LIN {X 0,Y 474.686,Z 210.351,A -85,B 0,C 180,E1 -7391.963,E2 -7391.963} C_VEL
LIN {X 0,Y 474.649,Z 210.356,A -85,B 0,C 180,E1 -7395.778,E2 -7395.778} C_VEL
LIN {X 0,Y 474.614,Z 210.365,A -85,B 0,C 180,E1 -7399.012,E2 -7399.012} C_VEL
LIN {X 0,Y 474.547,Z 210.369,A -85,B 0,C 180,E1 -7401.731,E2 -7401.731} C_VEL
LIN {X 0,Y 474.613,Z 210.367,A -85,B 0,C 180,E1 -7404.495,E2 -7404.495} C_VEL
LIN {X 0,Y 474.635,Z 210.358,A -85,B 0,C 180,E1 -7407.337,E2 -7407.337} C_VEL
LIN {X 0,Y 474.56,Z 210.372,A -85,B 0,C 180,E1 -7410.813,E2 -7410.813} C_VEL
LIN {X 0,Y 474.597,Z 210.364,A -85,B 0,C 180,E1 -7413.987,E2 -7413.987} C_VEL
LIN {X 0,Y 474.534,Z 210.373,A -85,B 0,C 180,E1 -7416.903,E2 -7416.903} C_VEL
LIN {X 0,Y 474.58,Z 210.365,A -85,B 0,C 180,E1 -7419.649,E2 -7419.649} C_VEL
LIN {X 0,Y 474.589,Z 210.37,A -85,B 0,C 180,E1 -7422.24,E2 -7422.24} C_VEL
LIN {X 0,Y 474.584,Z 210.364,A -85,B 0,C 180,E1 -7425.301,E2 -7425.301} C_VEL
LIN {X 0,Y 474.591,Z 210.371,A -85,B 0,C 180,E1 -7428.218,E2 -7428.218} C_VEL
LIN {X 0,Y 474.617,Z 210.365,A -85,B 0,C 180,E1 -7430.458,E2 -7430.458} C_VEL
LIN {X 0,Y 474.568,Z 210.368,A -85,B 0,C 180,E1 -7433.68,E2 -7433.68} C_VEL
LIN {X 0,Y 474.621,Z 210.36,A -85,B 0,C 180,E1 -7436.783,E2 -7436.783} C_VEL
LIN {X 0,Y 474.586,Z 210.368,A -85,B 0,C 180,E1 -7439.773,E2 -7439.773} C_VEL
LIN {X 0,Y 474.681,Z 210.353,A -85,B 0,C 180,E1 -7442.683,E2 -7442.683} C_VEL
LIN {X 0,Y 474.627,Z 210.361,A -85,B 0,C 180,E1 -7445.509,E2 -7445.509} C_VEL
LIN {X 0,Y 474.659,Z 210.355,A -85,B 0,C 180,E1 -7449.188,E2 -7449.188} C_VEL
LIN {X 0,Y 474.634,Z 210.363,A -85,B 0,C 180,E1 -7451.707,E2 -7451.707} C_VEL
LIN {X 0,Y 473.967,Z 210.452,A -85,B 0,C 180,E1 -7452.416,E2 -7452.416} C_VEL
LIN {X 0,Y 471.117,Z 210.806,A -85,B 0,C 180,E1 -7453.568,E2 -7453.568} C_VEL
LIN {X 0,Y 468.706,Z 211.101,A -85,B 0,C 180,E1 -7454.496,E2 -7454.496} C_VEL
LIN {X 0,Y 467.669,Z 211.227,A -85,B 0,C 180,E1 -7455.213,E2 -7455.213} C_VEL
LIN {X 0,Y 467.583,Z 211.237,A -85,B 0,C 180,E1 -7455.456,E2 -7455.456} C_VEL
LIN {X 0,Y 467.645,Z 211.228,A -85,B 0,C 180,E1 -7458.736,E2 -7458.736} C_VEL
LIN {X 0,Y 467.666,Z 211.23,A -85,B 0,C 180,E1 -7461.359,E2 -7461.359} C_VEL
LIN {X 0,Y 467.718,Z 211.227,A -85,B 0,C 180,E1 -7463.964,E2 -7463.964} C_VEL
LIN {X 0,Y 467.696,Z 211.354,A -85,B 0,C 180,E1 -7465.099,E2 -7465.099} C_VEL
LIN {X 0,Y 468.519,Z 218.325,A -85,B 0,C 180,E1 -7466.562,E2 -7466.562} C_VEL
LIN {X 0,Y 468.443,Z 226.016,A -85,B 0,C 180,E1 -7468.121,E2 -7468.121} C_VEL
LIN {X 0,Y 471.287,Z 240.784,A -85,B 0,C 180,E1 -7468.453,E2 -7468.453} C_VEL
LIN {X 0,Y 470.521,Z 333.446,A -85,B 0,C 180,E1 -7469.895,E2 -7469.895} C_VEL
LIN {X 0,Y 470.229,Z 346.46,A -85,B 0,C 180,E1 -7470.269,E2 -7470.269} C_VEL
LIN {X 0,Y 469.945,Z 358.958,A -85,B 0,C 180,E1 -7470.805,E2 -7470.805} C_VEL
LIN {X 0,Y 469.51,Z 370.947,A -85,B 0,C 180,E1 -7471.502,E2 -7471.502} C_VEL
LIN {X 0,Y 468.954,Z 382.395,A -85,B 0,C 180,E1 -7472.363,E2 -7472.363} C_VEL
LIN {X 0,Y 468.529,Z 392.675,A -85,B 0,C 180,E1 -7473.333,E2 -7473.333} C_VEL
LIN {X 0,Y 468.097,Z 401.117,A -85,B 0,C 180,E1 -7474.306,E2 -7474.306} C_VEL
LIN {X 0,Y 467.694,Z 410.256,A -85,B 0,C 180,E1 -7475.606,E2 -7475.606} C_VEL
LIN {X 0,Y 467.398,Z 417.615,A -85,B 0,C 180,E1 -7476.91,E2 -7476.91} C_VEL
LIN {X 0,Y 467.126,Z 423.538,A -85,B 0,C 180,E1 -7478.218,E2 -7478.218} C_VEL
LIN {X 0,Y 466.911,Z 428.222,A -85,B 0,C 180,E1 -7479.531,E2 -7479.531} C_VEL
LIN {X 0,Y 466.795,Z 431.791,A -85,B 0,C 180,E1 -7480.848,E2 -7480.848} C_VEL
LIN {X 0,Y 466.701,Z 434.341,A -85,B 0,C 180,E1 -7482.171,E2 -7482.171} C_VEL
LIN {X 0,Y 466.604,Z 435.521,A -85,B 0,C 180,E1 -7483.058,E2 -7483.058} C_VEL
LIN {X 0,Y 466.58,Z 436.247,A -85,B 0,C 180,E1 -7483.946,E2 -7483.946} C_VEL
LIN {X 0,Y 466.616,Z 436.558,A -85,B 0,C 180,E1 -7485.433,E2 -7485.433} C_VEL
LIN {X 0,Y 466.566,Z 435.978,A -85,B 0,C 180,E1 -7486.631,E2 -7486.631} C_VEL
LIN {X 0,Y 466.628,Z 435.02,A -85,B 0,C 180,E1 -7487.531,E2 -7487.531} C_VEL
LIN {X 0,Y 466.737,Z 433.625,A -85,B 0,C 180,E1 -7488.444,E2 -7488.444} C_VEL
LIN {X 0,Y 466.862,Z 430.671,A -85,B 0,C 180,E1 -7489.798,E2 -7489.798} C_VEL
LIN {X 0,Y 467.026,Z 426.549,A -85,B 0,C 180,E1 -7491.171,E2 -7491.171} C_VEL
LIN {X 0,Y 467.303,Z 420.044,A -85,B 0,C 180,E1 -7492.784,E2 -7492.784} C_VEL
LIN {X 0,Y 467.679,Z 412.837,A -85,B 0,C 180,E1 -7494.172,E2 -7494.172} C_VEL
LIN {X 0,Y 468.058,Z 405.338,A -85,B 0,C 180,E1 -7495.336,E2 -7495.336} C_VEL
LIN {X 0,Y 468.534,Z 396.074,A -85,B 0,C 180,E1 -7496.502,E2 -7496.502} C_VEL
LIN {X 0,Y 469.022,Z 385.744,A -85,B 0,C 180,E1 -7497.557,E2 -7497.557} C_VEL
LIN {X 0,Y 469.553,Z 375.373,A -85,B 0,C 180,E1 -7498.407,E2 -7498.407} C_VEL
LIN {X 0,Y 470.036,Z 363.063,A -85,B 0,C 180,E1 -7499.196,E2 -7499.196} C_VEL
LIN {X 0,Y 470.43,Z 350.815,A -85,B 0,C 180,E1 -7499.784,E2 -7499.784} C_VEL
LIN {X 0,Y 470.664,Z 338.306,A -85,B 0,C 180,E1 -7500.211,E2 -7500.211} C_VEL
LIN {X 0,Y 470.823,Z 323.886,A -85,B 0,C 180,E1 -7500.497,E2 -7500.497} C_VEL
LIN {X 0,Y 471.613,Z 240.593,A -85,B 0,C 180,E1 -7501.782,E2 -7501.782} C_VEL
LIN {X 0,Y 468.664,Z 226.097,A -85,B 0,C 180,E1 -7502.147,E2 -7502.147} C_VEL
LIN {X 0,Y 468.703,Z 216.769,A -85,B 0,C 180,E1 -7504.025,E2 -7504.025} C_VEL
LIN {X 0,Y 467.613,Z 211.238,A -85,B 0,C 180,E1 -7505.221,E2 -7505.221} C_VEL
LIN {X 0,Y 467.564,Z 211.247,A -85,B 0,C 180,E1 -7508.592,E2 -7508.592} C_VEL
LIN {X 0,Y 467.577,Z 211.237,A -85,B 0,C 180,E1 -7511.4,E2 -7511.4} C_VEL
LIN {X 0,Y 467.561,Z 211.246,A -85,B 0,C 180,E1 -7513.822,E2 -7513.822} C_VEL
LIN {X 0,Y 467.595,Z 211.237,A -85,B 0,C 180,E1 -7517.441,E2 -7517.441} C_VEL
LIN {X 0,Y 467.581,Z 211.239,A -85,B 0,C 180,E1 -7520.856,E2 -7520.856} C_VEL
LIN {X 0,Y 467.543,Z 211.245,A -85,B 0,C 180,E1 -7524.259,E2 -7524.259} C_VEL
LIN {X 0,Y 467.561,Z 211.241,A -85,B 0,C 180,E1 -7527.32,E2 -7527.32} C_VEL
LIN {X 0,Y 467.553,Z 211.239,A -85,B 0,C 180,E1 -7530.665,E2 -7530.665} C_VEL
LIN {X 0,Y 467.592,Z 211.236,A -85,B 0,C 180,E1 -7533.198,E2 -7533.198} C_VEL
LIN {X 0,Y 467.573,Z 211.238,A -85,B 0,C 180,E1 -7536.466,E2 -7536.466} C_VEL
LIN {X 0,Y 467.598,Z 211.239,A -85,B 0,C 180,E1 -7539.776,E2 -7539.776} C_VEL
LIN {X 0,Y 467.584,Z 211.234,A -85,B 0,C 180,E1 -7542.506,E2 -7542.506} C_VEL
LIN {X 0,Y 467.579,Z 211.24,A -85,B 0,C 180,E1 -7545.196,E2 -7545.196} C_VEL
LIN {X 0,Y 467.626,Z 211.234,A -85,B 0,C 180,E1 -7547.854,E2 -7547.854} C_VEL
LIN {X 0,Y 467.653,Z 211.231,A -85,B 0,C 180,E1 -7551.357,E2 -7551.357} C_VEL
LIN {X 0,Y 467.725,Z 211.22,A -85,B 0,C 180,E1 -7553.963,E2 -7553.963} C_VEL
LIN {X 0,Y 467.827,Z 211.209,A -85,B 0,C 180,E1 -7557.417,E2 -7557.417} C_VEL
LIN {X 0,Y 467.846,Z 211.2,A -85,B 0,C 180,E1 -7560,E2 -7560} C_VEL
LIN {X 0,Y 467.826,Z 211.204,A -85,B 0,C 180,E1 -7562.583,E2 -7562.583} C_VEL
LIN {X 0,Y 467.697,Z 211.216,A -85,B 0,C 180,E1 -7566.038,E2 -7566.038} C_VEL
LIN {X 0,Y 467.64,Z 211.23,A -85,B 0,C 180,E1 -7568.644,E2 -7568.644} C_VEL
LIN {X 0,Y 467.654,Z 211.226,A -85,B 0,C 180,E1 -7572.146,E2 -7572.146} C_VEL
LIN {X 0,Y 467.62,Z 211.23,A -85,B 0,C 180,E1 -7575.885,E2 -7575.885} C_VEL
LIN {X 0,Y 467.594,Z 211.235,A -85,B 0,C 180,E1 -7579.309,E2 -7579.309} C_VEL
LIN {X 0,Y 467.504,Z 211.247,A -85,B 0,C 180,E1 -7582.076,E2 -7582.076} C_VEL
LIN {X 0,Y 467.542,Z 211.248,A -85,B 0,C 180,E1 -7584.891,E2 -7584.891} C_VEL
LIN {X 0,Y 467.557,Z 211.238,A -85,B 0,C 180,E1 -7587.773,E2 -7587.773} C_VEL
LIN {X 0,Y 467.529,Z 211.244,A -85,B 0,C 180,E1 -7591.043,E2 -7591.043} C_VEL
LIN {X 0,Y 467.557,Z 211.245,A -85,B 0,C 180,E1 -7594.242,E2 -7594.242} C_VEL
LIN {X 0,Y 467.523,Z 211.243,A -85,B 0,C 180,E1 -7597.187,E2 -7597.187} C_VEL
LIN {X 0,Y 467.554,Z 211.245,A -85,B 0,C 180,E1 -7600.267,E2 -7600.267} C_VEL
LIN {X 0,Y 467.547,Z 211.242,A -85,B 0,C 180,E1 -7602.565,E2 -7602.565} C_VEL
LIN {X 0,Y 467.553,Z 211.241,A -85,B 0,C 180,E1 -7605.054,E2 -7605.054} C_VEL
LIN {X 0,Y 467.557,Z 211.243,A -85,B 0,C 180,E1 -7608.598,E2 -7608.598} C_VEL
LIN {X 0,Y 467.556,Z 211.247,A -85,B 0,C 180,E1 -7611.957,E2 -7611.957} C_VEL
LIN {X 0,Y 467.559,Z 211.242,A -85,B 0,C 180,E1 -7615.169,E2 -7615.169} C_VEL
LIN {X 0,Y 467.579,Z 211.243,A -85,B 0,C 180,E1 -7618.261,E2 -7618.261} C_VEL
LIN {X 0,Y 467.553,Z 211.245,A -85,B 0,C 180,E1 -7621.25,E2 -7621.25} C_VEL
LIN {X 0,Y 467.62,Z 211.35,A -85,B 0,C 180,E1 -7623.412,E2 -7623.412} C_VEL
LIN {X 0,Y 469.92,Z 222.915,A -85,B 0,C 180,E1 -7625.584,E2 -7625.584} C_VEL
LIN {X 0,Y 469.761,Z 230.399,A -85,B 0,C 180,E1 -7626.877,E2 -7626.877} C_VEL
LIN {X 0,Y 468.999,Z 247.876,A -85,B 0,C 180,E1 -7629.839,E2 -7629.839} C_VEL
LIN {X 0,Y 468.318,Z 265.993,A -85,B 0,C 180,E1 -7632.868,E2 -7632.868} C_VEL
LIN {X 0,Y 471.329,Z 286.597,A -85,B 0,C 180,E1 -7633.336,E2 -7633.336} C_VEL
LIN {X 0,Y 470.643,Z 374.605,A -85,B 0,C 180,E1 -7634.713,E2 -7634.713} C_VEL
LIN {X 0,Y 470.245,Z 387.918,A -85,B 0,C 180,E1 -7635.088,E2 -7635.088} C_VEL
LIN {X 0,Y 469.71,Z 401.233,A -85,B 0,C 180,E1 -7635.652,E2 -7635.652} C_VEL
LIN {X 0,Y 469.193,Z 413.216,A -85,B 0,C 180,E1 -7636.354,E2 -7636.354} C_VEL
LIN {X 0,Y 468.661,Z 425.052,A -85,B 0,C 180,E1 -7637.251,E2 -7637.251} C_VEL
LIN {X 0,Y 468.137,Z 436.079,A -85,B 0,C 180,E1 -7638.306,E2 -7638.306} C_VEL
LIN {X 0,Y 467.662,Z 445.209,A -85,B 0,C 180,E1 -7639.391,E2 -7639.391} C_VEL
LIN {X 0,Y 467.246,Z 454.137,A -85,B 0,C 180,E1 -7640.694,E2 -7640.694} C_VEL
LIN {X 0,Y 466.988,Z 461.326,A -85,B 0,C 180,E1 -7641.997,E2 -7641.997} C_VEL
LIN {X 0,Y 466.832,Z 466.188,A -85,B 0,C 180,E1 -7643.082,E2 -7643.082} C_VEL
LIN {X 0,Y 466.728,Z 470.915,A -85,B 0,C 180,E1 -7644.382,E2 -7644.382} C_VEL
LIN {X 0,Y 466.648,Z 474.527,A -85,B 0,C 180,E1 -7645.68,E2 -7645.68} C_VEL
LIN {X 0,Y 466.692,Z 476.391,A -85,B 0,C 180,E1 -7646.545,E2 -7646.545} C_VEL
LIN {X 0,Y 466.68,Z 477.787,A -85,B 0,C 180,E1 -7647.409,E2 -7647.409} C_VEL
LIN {X 0,Y 466.661,Z 478.786,A -85,B 0,C 180,E1 -7648.273,E2 -7648.273} C_VEL
LIN {X 0,Y 466.624,Z 479.393,A -85,B 0,C 180,E1 -7649.136,E2 -7649.136} C_VEL
LIN {X 0,Y 466.607,Z 479.602,A -85,B 0,C 180,E1 -7649.999,E2 -7649.999} C_VEL
LIN {X 0,Y 466.661,Z 478.765,A -85,B 0,C 180,E1 -7651.724,E2 -7651.724} C_VEL
LIN {X 0,Y 466.68,Z 477.76,A -85,B 0,C 180,E1 -7652.588,E2 -7652.588} C_VEL
LIN {X 0,Y 466.691,Z 476.344,A -85,B 0,C 180,E1 -7653.452,E2 -7653.452} C_VEL
LIN {X 0,Y 466.687,Z 473.377,A -85,B 0,C 180,E1 -7654.749,E2 -7654.749} C_VEL
LIN {X 0,Y 466.741,Z 469.359,A -85,B 0,C 180,E1 -7656.048,E2 -7656.048} C_VEL
LIN {X 0,Y 466.9,Z 463.172,A -85,B 0,C 180,E1 -7657.566,E2 -7657.566} C_VEL
LIN {X 0,Y 467.123,Z 456.421,A -85,B 0,C 180,E1 -7658.869,E2 -7658.869} C_VEL
LIN {X 0,Y 467.448,Z 448.044,A -85,B 0,C 180,E1 -7660.173,E2 -7660.173} C_VEL
LIN {X 0,Y 467.896,Z 439.429,A -85,B 0,C 180,E1 -7661.258,E2 -7661.258} C_VEL
LIN {X 0,Y 468.335,Z 429.329,A -85,B 0,C 180,E1 -7662.295,E2 -7662.295} C_VEL
LIN {X 0,Y 468.864,Z 418.26,A -85,B 0,C 180,E1 -7663.211,E2 -7663.211} C_VEL
LIN {X 0,Y 469.325,Z 406.612,A -85,B 0,C 180,E1 -7663.97,E2 -7663.97} C_VEL
LIN {X 0,Y 469.801,Z 394.509,A -85,B 0,C 180,E1 -7664.564,E2 -7664.564} C_VEL
LIN {X 0,Y 470.205,Z 381.375,A -85,B 0,C 180,E1 -7665.021,E2 -7665.021} C_VEL
LIN {X 0,Y 470.528,Z 368.86,A -85,B 0,C 180,E1 -7665.288,E2 -7665.288} C_VEL
LIN {X 0,Y 470.904,Z 284.953,A -85,B 0,C 180,E1 -7666.579,E2 -7666.579} C_VEL
LIN {X 0,Y 468.244,Z 266.3,A -85,B 0,C 180,E1 -7666.984,E2 -7666.984} C_VEL
LIN {X 0,Y 468.862,Z 248.509,A -85,B 0,C 180,E1 -7669.935,E2 -7669.935} C_VEL
LIN {X 0,Y 469.653,Z 229.451,A -85,B 0,C 180,E1 -7673.126,E2 -7673.126} C_VEL
LIN {X 0,Y 469.698,Z 221.967,A -85,B 0,C 180,E1 -7674.403,E2 -7674.403} C_VEL
LIN {X 0,Y 467.671,Z 211.233,A -85,B 0,C 180,E1 -7676.371,E2 -7676.371} C_VEL
LIN {X 0,Y 467.539,Z 211.249,A -85,B 0,C 180,E1 -7679.734,E2 -7679.734} C_VEL
LIN {X 0,Y 467.567,Z 211.239,A -85,B 0,C 180,E1 -7682.754,E2 -7682.754} C_VEL
LIN {X 0,Y 467.537,Z 211.249,A -85,B 0,C 180,E1 -7685.885,E2 -7685.885} C_VEL
LIN {X 0,Y 467.559,Z 211.239,A -85,B 0,C 180,E1 -7689.141,E2 -7689.141} C_VEL
LIN {X 0,Y 467.561,Z 211.24,A -85,B 0,C 180,E1 -7692.563,E2 -7692.563} C_VEL
LIN {X 0,Y 467.544,Z 211.245,A -85,B 0,C 180,E1 -7696.173,E2 -7696.173} C_VEL
LIN {X 0,Y 467.559,Z 211.239,A -85,B 0,C 180,E1 -7698.718,E2 -7698.718} C_VEL
LIN {X 0,Y 467.544,Z 211.245,A -85,B 0,C 180,E1 -7701.403,E2 -7701.403} C_VEL
LIN {X 0,Y 467.526,Z 211.245,A -85,B 0,C 180,E1 -7704.257,E2 -7704.257} C_VEL
LIN {X 0,Y 467.543,Z 211.245,A -85,B 0,C 180,E1 -7707.317,E2 -7707.317} C_VEL
LIN {X 0,Y 467.536,Z 211.242,A -85,B 0,C 180,E1 -7710.663,E2 -7710.663} C_VEL
LIN {X 0,Y 467.576,Z 211.241,A -85,B 0,C 180,E1 -7713.197,E2 -7713.197} C_VEL
LIN {X 0,Y 467.541,Z 211.243,A -85,B 0,C 180,E1 -7716.055,E2 -7716.055} C_VEL
LIN {X 0,Y 467.593,Z 211.236,A -85,B 0,C 180,E1 -7718.855,E2 -7718.855} C_VEL
LIN {X 0,Y 467.583,Z 211.241,A -85,B 0,C 180,E1 -7721.6,E2 -7721.6} C_VEL
LIN {X 0,Y 467.605,Z 211.233,A -85,B 0,C 180,E1 -7724.304,E2 -7724.304} C_VEL
LIN {X 0,Y 467.646,Z 211.23,A -85,B 0,C 180,E1 -7727.854,E2 -7727.854} C_VEL
LIN {X 0,Y 467.644,Z 211.235,A -85,B 0,C 180,E1 -7731.356,E2 -7731.356} C_VEL
LIN {X 0,Y 467.708,Z 211.221,A -85,B 0,C 180,E1 -7733.962,E2 -7733.962} C_VEL
LIN {X 0,Y 467.806,Z 211.213,A -85,B 0,C 180,E1 -7737.417,E2 -7737.417} C_VEL
LIN {X 0,Y 467.824,Z 211.206,A -85,B 0,C 180,E1 -7740,E2 -7740} C_VEL
LIN {X 0,Y 467.805,Z 211.211,A -85,B 0,C 180,E1 -7742.583,E2 -7742.583} C_VEL
LIN {X 0,Y 467.682,Z 211.224,A -85,B 0,C 180,E1 -7746.038,E2 -7746.038} C_VEL
LIN {X 0,Y 467.629,Z 211.235,A -85,B 0,C 180,E1 -7748.643,E2 -7748.643} C_VEL
LIN {X 0,Y 467.63,Z 211.231,A -85,B 0,C 180,E1 -7752.146,E2 -7752.146} C_VEL
LIN {X 0,Y 467.615,Z 211.232,A -85,B 0,C 180,E1 -7755.894,E2 -7755.894} C_VEL
LIN {X 0,Y 467.573,Z 211.239,A -85,B 0,C 180,E1 -7759.31,E2 -7759.31} C_VEL
LIN {X 0,Y 467.492,Z 211.249,A -85,B 0,C 180,E1 -7762.076,E2 -7762.076} C_VEL
LIN {X 0,Y 467.557,Z 211.244,A -85,B 0,C 180,E1 -7764.89,E2 -7764.89} C_VEL
LIN {X 0,Y 467.574,Z 211.237,A -85,B 0,C 180,E1 -7767.772,E2 -7767.772} C_VEL
LIN {X 0,Y 467.524,Z 211.246,A -85,B 0,C 180,E1 -7771.048,E2 -7771.048} C_VEL
LIN {X 0,Y 467.549,Z 211.245,A -85,B 0,C 180,E1 -7774.245,E2 -7774.245} C_VEL
LIN {X 0,Y 467.51,Z 211.246,A -85,B 0,C 180,E1 -7777.19,E2 -7777.19} C_VEL
LIN {X 0,Y 467.538,Z 211.248,A -85,B 0,C 180,E1 -7780.268,E2 -7780.268} C_VEL
LIN {X 0,Y 467.553,Z 211.245,A -85,B 0,C 180,E1 -7782.57,E2 -7782.57} C_VEL
LIN {X 0,Y 467.533,Z 211.243,A -85,B 0,C 180,E1 -7785.056,E2 -7785.056} C_VEL
LIN {X 0,Y 467.56,Z 211.239,A -85,B 0,C 180,E1 -7787.444,E2 -7787.444} C_VEL
LIN {X 0,Y 467.555,Z 211.241,A -85,B 0,C 180,E1 -7790.859,E2 -7790.859} C_VEL
LIN {X 0,Y 467.539,Z 211.248,A -85,B 0,C 180,E1 -7794.264,E2 -7794.264} C_VEL
LIN {X 0,Y 467.561,Z 211.239,A -85,B 0,C 180,E1 -7797.325,E2 -7797.325} C_VEL
LIN {X 0,Y 467.551,Z 211.241,A -85,B 0,C 180,E1 -7800.671,E2 -7800.671} C_VEL
LIN {X 0,Y 467.597,Z 211.235,A -85,B 0,C 180,E1 -7803.203,E2 -7803.203} C_VEL
LIN {X 0,Y 467.578,Z 211.239,A -85,B 0,C 180,E1 -7806.472,E2 -7806.472} C_VEL
LIN {X 0,Y 467.61,Z 211.24,A -85,B 0,C 180,E1 -7809.78,E2 -7809.78} C_VEL
LIN {X 0,Y 467.585,Z 211.237,A -85,B 0,C 180,E1 -7812.509,E2 -7812.509} C_VEL
LIN {X 0,Y 467.593,Z 211.236,A -85,B 0,C 180,E1 -7815.199,E2 -7815.199} C_VEL
LIN {X 0,Y 467.583,Z 211.237,A -85,B 0,C 180,E1 -7815.456,E2 -7815.456} C_VEL
LIN {X 0,Y 466.916,Z 211.323,A -85,B 0,C 180,E1 -7816.176,E2 -7816.176} C_VEL
LIN {X 0,Y 464.073,Z 211.676,A -85,B 0,C 180,E1 -7817.344,E2 -7817.344} C_VEL
LIN {X 0,Y 461.674,Z 211.974,A -85,B 0,C 180,E1 -7818.286,E2 -7818.286} C_VEL
LIN {X 0,Y 460.649,Z 212.101,A -85,B 0,C 180,E1 -7819.014,E2 -7819.014} C_VEL
LIN {X 0,Y 460.567,Z 212.113,A -85,B 0,C 180,E1 -7819.26,E2 -7819.26} C_VEL
LIN {X 0,Y 460.665,Z 212.102,A -85,B 0,C 180,E1 -7822.59,E2 -7822.59} C_VEL
LIN {X 0,Y 460.68,Z 212.192,A -85,B 0,C 180,E1 -7824.942,E2 -7824.942} C_VEL
LIN {X 0,Y 461.538,Z 219.578,A -85,B 0,C 180,E1 -7826.51,E2 -7826.51} C_VEL
LIN {X 0,Y 461.48,Z 226.212,A -85,B 0,C 180,E1 -7827.863,E2 -7827.863} C_VEL
LIN {X 0,Y 464.439,Z 241.12,A -85,B 0,C 180,E1 -7828.223,E2 -7828.223} C_VEL
LIN {X 0,Y 463.664,Z 333.274,A -85,B 0,C 180,E1 -7829.676,E2 -7829.676} C_VEL
LIN {X 0,Y 463.384,Z 345.702,A -85,B 0,C 180,E1 -7830.029,E2 -7830.029} C_VEL
LIN {X 0,Y 463.044,Z 359.049,A -85,B 0,C 180,E1 -7830.599,E2 -7830.599} C_VEL
LIN {X 0,Y 462.604,Z 371.1,A -85,B 0,C 180,E1 -7831.307,E2 -7831.307} C_VEL
LIN {X 0,Y 462.024,Z 382.58,A -85,B 0,C 180,E1 -7832.181,E2 -7832.181} C_VEL
LIN {X 0,Y 461.552,Z 392.892,A -85,B 0,C 180,E1 -7833.165,E2 -7833.165} C_VEL
LIN {X 0,Y 461.117,Z 401.347,A -85,B 0,C 180,E1 -7834.153,E2 -7834.153} C_VEL
LIN {X 0,Y 460.793,Z 409.135,A -85,B 0,C 180,E1 -7835.252,E2 -7835.252} C_VEL
LIN {X 0,Y 460.402,Z 416.772,A -85,B 0,C 180,E1 -7836.575,E2 -7836.575} C_VEL
LIN {X 0,Y 460.105,Z 422.916,A -85,B 0,C 180,E1 -7837.902,E2 -7837.902} C_VEL
LIN {X 0,Y 459.885,Z 427.798,A -85,B 0,C 180,E1 -7839.234,E2 -7839.234} C_VEL
LIN {X 0,Y 459.741,Z 431.556,A -85,B 0,C 180,E1 -7840.571,E2 -7840.571} C_VEL
LIN {X 0,Y 459.652,Z 434.245,A -85,B 0,C 180,E1 -7841.89,E2 -7841.89} C_VEL
LIN {X 0,Y 459.525,Z 436.044,A -85,B 0,C 180,E1 -7843.263,E2 -7843.263} C_VEL
LIN {X 0,Y 459.496,Z 436.693,A -85,B 0,C 180,E1 -7844.166,E2 -7844.166} C_VEL
LIN {X 0,Y 459.521,Z 436.875,A -85,B 0,C 180,E1 -7845.522,E2 -7845.522} C_VEL
LIN {X 0,Y 459.508,Z 436.108,A -85,B 0,C 180,E1 -7846.894,E2 -7846.894} C_VEL
LIN {X 0,Y 459.658,Z 433.871,A -85,B 0,C 180,E1 -7848.567,E2 -7848.567} C_VEL
LIN {X 0,Y 459.807,Z 430.414,A -85,B 0,C 180,E1 -7850.115,E2 -7850.115} C_VEL
LIN {X 0,Y 460,Z 426.081,A -85,B 0,C 180,E1 -7851.51,E2 -7851.51} C_VEL
LIN {X 0,Y 460.274,Z 420.419,A -85,B 0,C 180,E1 -7852.914,E2 -7852.914} C_VEL
LIN {X 0,Y 460.694,Z 413.224,A -85,B 0,C 180,E1 -7854.323,E2 -7854.323} C_VEL
LIN {X 0,Y 461.175,Z 404.553,A -85,B 0,C 180,E1 -7855.666,E2 -7855.666} C_VEL
LIN {X 0,Y 461.649,Z 395.45,A -85,B 0,C 180,E1 -7856.807,E2 -7856.807} C_VEL
LIN {X 0,Y 462.216,Z 384.923,A -85,B 0,C 180,E1 -7857.875,E2 -7857.875} C_VEL
LIN {X 0,Y 462.833,Z 373.327,A -85,B 0,C 180,E1 -7858.798,E2 -7858.798} C_VEL
LIN {X 0,Y 463.299,Z 361.462,A -85,B 0,C 180,E1 -7859.537,E2 -7859.537} C_VEL
LIN {X 0,Y 463.646,Z 350.086,A -85,B 0,C 180,E1 -7860.074,E2 -7860.074} C_VEL
LIN {X 0,Y 463.908,Z 337.621,A -85,B 0,C 180,E1 -7860.486,E2 -7860.486} C_VEL
LIN {X 0,Y 464.124,Z 320.907,A -85,B 0,C 180,E1 -7860.802,E2 -7860.802} C_VEL
LIN {X 0,Y 464.804,Z 240.939,A -85,B 0,C 180,E1 -7862.062,E2 -7862.062} C_VEL
LIN {X 0,Y 461.74,Z 226.372,A -85,B 0,C 180,E1 -7862.449,E2 -7862.449} C_VEL
LIN {X 0,Y 461.805,Z 218.708,A -85,B 0,C 180,E1 -7864.004,E2 -7864.004} C_VEL
LIN {X 0,Y 460.554,Z 212.117,A -85,B 0,C 180,E1 -7865.44,E2 -7865.44} C_VEL
LIN {X 0,Y 460.548,Z 212.119,A -85,B 0,C 180,E1 -7868.898,E2 -7868.898} C_VEL
LIN {X 0,Y 460.536,Z 212.118,A -85,B 0,C 180,E1 -7872.177,E2 -7872.177} C_VEL
LIN {X 0,Y 460.507,Z 212.121,A -85,B 0,C 180,E1 -7875.411,E2 -7875.411} C_VEL
LIN {X 0,Y 460.527,Z 212.122,A -85,B 0,C 180,E1 -7878.395,E2 -7878.395} C_VEL
LIN {X 0,Y 460.521,Z 212.118,A -85,B 0,C 180,E1 -7881.267,E2 -7881.267} C_VEL
LIN {X 0,Y 460.493,Z 212.12,A -85,B 0,C 180,E1 -7884.553,E2 -7884.553} C_VEL
LIN {X 0,Y 460.511,Z 212.122,A -85,B 0,C 180,E1 -7887.714,E2 -7887.714} C_VEL
LIN {X 0,Y 460.523,Z 212.114,A -85,B 0,C 180,E1 -7890.768,E2 -7890.768} C_VEL
LIN {X 0,Y 460.539,Z 212.12,A -85,B 0,C 180,E1 -7893.734,E2 -7893.734} C_VEL
LIN {X 0,Y 460.527,Z 212.115,A -85,B 0,C 180,E1 -7896.623,E2 -7896.623} C_VEL
LIN {X 0,Y 460.546,Z 212.113,A -85,B 0,C 180,E1 -7899.453,E2 -7899.453} C_VEL
LIN {X 0,Y 460.533,Z 212.113,A -85,B 0,C 180,E1 -7902.229,E2 -7902.229} C_VEL
LIN {X 0,Y 460.542,Z 212.115,A -85,B 0,C 180,E1 -7904.964,E2 -7904.964} C_VEL
LIN {X 0,Y 460.583,Z 212.108,A -85,B 0,C 180,E1 -7908.559,E2 -7908.559} C_VEL
LIN {X 0,Y 460.667,Z 212.095,A -85,B 0,C 180,E1 -7912.108,E2 -7912.108} C_VEL
LIN {X 0,Y 460.672,Z 212.098,A -85,B 0,C 180,E1 -7914.748,E2 -7914.748} C_VEL
LIN {X 0,Y 460.768,Z 212.087,A -85,B 0,C 180,E1 -7917.378,E2 -7917.378} C_VEL
LIN {X 0,Y 460.818,Z 212.076,A -85,B 0,C 180,E1 -7920,E2 -7920} C_VEL
LIN {X 0,Y 460.767,Z 212.083,A -85,B 0,C 180,E1 -7922.623,E2 -7922.623} C_VEL
LIN {X 0,Y 460.662,Z 212.092,A -85,B 0,C 180,E1 -7926.131,E2 -7926.131} C_VEL
LIN {X 0,Y 460.591,Z 212.11,A -85,B 0,C 180,E1 -7928.777,E2 -7928.777} C_VEL
LIN {X 0,Y 460.607,Z 212.105,A -85,B 0,C 180,E1 -7932.458,E2 -7932.458} C_VEL
LIN {X 0,Y 460.574,Z 212.108,A -85,B 0,C 180,E1 -7935.999,E2 -7935.999} C_VEL
LIN {X 0,Y 460.541,Z 212.112,A -85,B 0,C 180,E1 -7939.617,E2 -7939.617} C_VEL
LIN {X 0,Y 460.481,Z 212.125,A -85,B 0,C 180,E1 -7942.43,E2 -7942.43} C_VEL
LIN {X 0,Y 460.523,Z 212.117,A -85,B 0,C 180,E1 -7945.798,E2 -7945.798} C_VEL
LIN {X 0,Y 460.504,Z 212.119,A -85,B 0,C 180,E1 -7948.237,E2 -7948.237} C_VEL
LIN {X 0,Y 460.5,Z 212.118,A -85,B 0,C 180,E1 -7951.284,E2 -7951.284} C_VEL
LIN {X 0,Y 460.502,Z 212.123,A -85,B 0,C 180,E1 -7954.505,E2 -7954.505} C_VEL
LIN {X 0,Y 460.481,Z 212.12,A -85,B 0,C 180,E1 -7957.625,E2 -7957.625} C_VEL
LIN {X 0,Y 460.513,Z 212.112,A -85,B 0,C 180,E1 -7961.014,E2 -7961.014} C_VEL
LIN {X 0,Y 460.5,Z 212.123,A -85,B 0,C 180,E1 -7964.591,E2 -7964.591} C_VEL
LIN {X 0,Y 460.492,Z 212.124,A -85,B 0,C 180,E1 -7967.818,E2 -7967.818} C_VEL
LIN {X 0,Y 460.504,Z 212.12,A -85,B 0,C 180,E1 -7970.137,E2 -7970.137} C_VEL
LIN {X 0,Y 460.47,Z 212.122,A -85,B 0,C 180,E1 -7973.472,E2 -7973.472} C_VEL
LIN {X 0,Y 460.525,Z 212.12,A -85,B 0,C 180,E1 -7976.676,E2 -7976.676} C_VEL
LIN {X 0,Y 460.504,Z 212.123,A -85,B 0,C 180,E1 -7979.761,E2 -7979.761} C_VEL
LIN {X 0,Y 460.558,Z 212.239,A -85,B 0,C 180,E1 -7983.155,E2 -7983.155} C_VEL
LIN {X 0,Y 462.867,Z 223.553,A -85,B 0,C 180,E1 -7985.324,E2 -7985.324} C_VEL
LIN {X 0,Y 463.086,Z 227.57,A -85,B 0,C 180,E1 -7986.049,E2 -7986.049} C_VEL
LIN {X 0,Y 462.202,Z 245.022,A -85,B 0,C 180,E1 -7989.064,E2 -7989.064} C_VEL
LIN {X 0,Y 461.492,Z 262.475,A -85,B 0,C 180,E1 -7992.038,E2 -7992.038} C_VEL
LIN {X 0,Y 461.35,Z 265.769,A -85,B 0,C 180,E1 -7992.595,E2 -7992.595} C_VEL
LIN {X 0,Y 464.507,Z 286.405,A -85,B 0,C 180,E1 -7993.062,E2 -7993.062} C_VEL
LIN {X 0,Y 463.812,Z 375.134,A -85,B 0,C 180,E1 -7994.482,E2 -7994.482} C_VEL
LIN {X 0,Y 463.37,Z 388.914,A -85,B 0,C 180,E1 -7994.889,E2 -7994.889} C_VEL
LIN {X 0,Y 462.829,Z 401.302,A -85,B 0,C 180,E1 -7995.434,E2 -7995.434} C_VEL
LIN {X 0,Y 462.306,Z 413.177,A -85,B 0,C 180,E1 -7996.147,E2 -7996.147} C_VEL
LIN {X 0,Y 461.723,Z 424.959,A -85,B 0,C 180,E1 -7997.056,E2 -7997.056} C_VEL
LIN {X 0,Y 461.174,Z 435.928,A -85,B 0,C 180,E1 -7998.127,E2 -7998.127} C_VEL
LIN {X 0,Y 460.636,Z 445.027,A -85,B 0,C 180,E1 -7999.228,E2 -7999.228} C_VEL
LIN {X 0,Y 460.197,Z 453.921,A -85,B 0,C 180,E1 -8000.55,E2 -8000.55} C_VEL
LIN {X 0,Y 459.92,Z 461.075,A -85,B 0,C 180,E1 -8001.873,E2 -8001.873} C_VEL
LIN {X 0,Y 459.71,Z 467.609,A -85,B 0,C 180,E1 -8003.416,E2 -8003.416} C_VEL
LIN {X 0,Y 459.641,Z 471.935,A -85,B 0,C 180,E1 -8004.735,E2 -8004.735} C_VEL
LIN {X 0,Y 459.566,Z 474.23,A -85,B 0,C 180,E1 -8005.614,E2 -8005.614} C_VEL
LIN {X 0,Y 459.588,Z 476.083,A -85,B 0,C 180,E1 -8006.492,E2 -8006.492} C_VEL
LIN {X 0,Y 459.601,Z 477.476,A -85,B 0,C 180,E1 -8007.369,E2 -8007.369} C_VEL
LIN {X 0,Y 459.557,Z 479.074,A -85,B 0,C 180,E1 -8009.122,E2 -8009.122} C_VEL
LIN {X 0,Y 459.538,Z 479.275,A -85,B 0,C 180,E1 -8009.998,E2 -8009.998} C_VEL
LIN {X 0,Y 459.557,Z 479.045,A -85,B 0,C 180,E1 -8010.875,E2 -8010.875} C_VEL
LIN {X 0,Y 459.6,Z 477.417,A -85,B 0,C 180,E1 -8012.628,E2 -8012.628} C_VEL
LIN {X 0,Y 459.589,Z 475.991,A -85,B 0,C 180,E1 -8013.505,E2 -8013.505} C_VEL
LIN {X 0,Y 459.618,Z 473.016,A -85,B 0,C 180,E1 -8014.822,E2 -8014.822} C_VEL
LIN {X 0,Y 459.691,Z 468.024,A -85,B 0,C 180,E1 -8016.405,E2 -8016.405} C_VEL
LIN {X 0,Y 459.871,Z 461.757,A -85,B 0,C 180,E1 -8017.903,E2 -8017.903} C_VEL
LIN {X 0,Y 460.134,Z 454.75,A -85,B 0,C 180,E1 -8019.226,E2 -8019.226} C_VEL
LIN {X 0,Y 460.499,Z 445.958,A -85,B 0,C 180,E1 -8020.55,E2 -8020.55} C_VEL
LIN {X 0,Y 461.059,Z 435.976,A -85,B 0,C 180,E1 -8021.761,E2 -8021.761} C_VEL
LIN {X 0,Y 461.56,Z 425.208,A -85,B 0,C 180,E1 -8022.806,E2 -8022.806} C_VEL
LIN {X 0,Y 462.117,Z 412.956,A -85,B 0,C 180,E1 -8023.744,E2 -8023.744} C_VEL
LIN {X 0,Y 462.623,Z 400.796,A -85,B 0,C 180,E1 -8024.458,E2 -8024.458} C_VEL
LIN {X 0,Y 463.099,Z 387.253,A -85,B 0,C 180,E1 -8025.032,E2 -8025.032} C_VEL
LIN {X 0,Y 463.467,Z 374.717,A -85,B 0,C 180,E1 -8025.386,E2 -8025.386} C_VEL
LIN {X 0,Y 464.143,Z 286.299,A -85,B 0,C 180,E1 -8026.779,E2 -8026.779} C_VEL
LIN {X 0,Y 461.254,Z 265.979,A -85,B 0,C 180,E1 -8027.226,E2 -8027.226} C_VEL
LIN {X 0,Y 461.847,Z 249.376,A -85,B 0,C 180,E1 -8030.019,E2 -8030.019} C_VEL
LIN {X 0,Y 462.696,Z 230.314,A -85,B 0,C 180,E1 -8033.257,E2 -8033.257} C_VEL
LIN {X 0,Y 462.842,Z 224.003,A -85,B 0,C 180,E1 -8034.346,E2 -8034.346} C_VEL
LIN {X 0,Y 460.63,Z 212.11,A -85,B 0,C 180,E1 -8036.562,E2 -8036.562} C_VEL
LIN {X 0,Y 460.517,Z 212.123,A -85,B 0,C 180,E1 -8039.554,E2 -8039.554} C_VEL
LIN {X 0,Y 460.515,Z 212.122,A -85,B 0,C 180,E1 -8042.281,E2 -8042.281} C_VEL
LIN {X 0,Y 460.494,Z 212.121,A -85,B 0,C 180,E1 -8045.441,E2 -8045.441} C_VEL
LIN {X 0,Y 460.522,Z 212.116,A -85,B 0,C 180,E1 -8048.894,E2 -8048.894} C_VEL
LIN {X 0,Y 460.497,Z 212.123,A -85,B 0,C 180,E1 -8052.177,E2 -8052.177} C_VEL
LIN {X 0,Y 460.493,Z 212.122,A -85,B 0,C 180,E1 -8055.408,E2 -8055.408} C_VEL
LIN {X 0,Y 460.515,Z 212.118,A -85,B 0,C 180,E1 -8058.392,E2 -8058.392} C_VEL
LIN {X 0,Y 460.515,Z 212.119,A -85,B 0,C 180,E1 -8061.265,E2 -8061.265} C_VEL
LIN {X 0,Y 460.476,Z 212.122,A -85,B 0,C 180,E1 -8064.551,E2 -8064.551} C_VEL
LIN {X 0,Y 460.492,Z 212.126,A -85,B 0,C 180,E1 -8067.712,E2 -8067.712} C_VEL
LIN {X 0,Y 460.505,Z 212.118,A -85,B 0,C 180,E1 -8070.766,E2 -8070.766} C_VEL
LIN {X 0,Y 460.524,Z 212.121,A -85,B 0,C 180,E1 -8073.732,E2 -8073.732} C_VEL
LIN {X 0,Y 460.515,Z 212.117,A -85,B 0,C 180,E1 -8076.622,E2 -8076.622} C_VEL
LIN {X 0,Y 460.525,Z 212.123,A -85,B 0,C 180,E1 -8079.451,E2 -8079.451} C_VEL
LIN {X 0,Y 460.512,Z 212.117,A -85,B 0,C 180,E1 -8082.228,E2 -8082.228} C_VEL
LIN {X 0,Y 460.521,Z 212.119,A -85,B 0,C 180,E1 -8084.963,E2 -8084.963} C_VEL
LIN {X 0,Y 460.607,Z 212.108,A -85,B 0,C 180,E1 -8087.666,E2 -8087.666} C_VEL
LIN {X 0,Y 460.612,Z 212.113,A -85,B 0,C 180,E1 -8091.223,E2 -8091.223} C_VEL
LIN {X 0,Y 460.674,Z 212.098,A -85,B 0,C 180,E1 -8093.869,E2 -8093.869} C_VEL
LIN {X 0,Y 460.771,Z 212.089,A -85,B 0,C 180,E1 -8097.377,E2 -8097.377} C_VEL
LIN {X 0,Y 460.795,Z 212.082,A -85,B 0,C 180,E1 -8100,E2 -8100} C_VEL
LIN {X 0,Y 460.746,Z 212.091,A -85,B 0,C 180,E1 -8102.623,E2 -8102.623} C_VEL
LIN {X 0,Y 460.648,Z 212.1,A -85,B 0,C 180,E1 -8106.13,E2 -8106.13} C_VEL
LIN {X 0,Y 460.576,Z 212.115,A -85,B 0,C 180,E1 -8108.777,E2 -8108.777} C_VEL
LIN {X 0,Y 460.583,Z 212.111,A -85,B 0,C 180,E1 -8112.458,E2 -8112.458} C_VEL
LIN {X 0,Y 460.572,Z 212.11,A -85,B 0,C 180,E1 -8116.009,E2 -8116.009} C_VEL
LIN {X 0,Y 460.518,Z 212.116,A -85,B 0,C 180,E1 -8119.617,E2 -8119.617} C_VEL
LIN {X 0,Y 460.467,Z 212.127,A -85,B 0,C 180,E1 -8122.431,E2 -8122.431} C_VEL
LIN {X 0,Y 460.521,Z 212.116,A -85,B 0,C 180,E1 -8125.804,E2 -8125.804} C_VEL
LIN {X 0,Y 460.507,Z 212.121,A -85,B 0,C 180,E1 -8128.236,E2 -8128.236} C_VEL
LIN {X 0,Y 460.477,Z 212.122,A -85,B 0,C 180,E1 -8131.285,E2 -8131.285} C_VEL
LIN {X 0,Y 460.493,Z 212.127,A -85,B 0,C 180,E1 -8134.509,E2 -8134.509} C_VEL
LIN {X 0,Y 460.463,Z 212.123,A -85,B 0,C 180,E1 -8137.626,E2 -8137.626} C_VEL
LIN {X 0,Y 460.502,Z 212.125,A -85,B 0,C 180,E1 -8140.272,E2 -8140.272} C_VEL
LIN {X 0,Y 460.463,Z 212.123,A -85,B 0,C 180,E1 -8143.379,E2 -8143.379} C_VEL
LIN {X 0,Y 460.465,Z 212.126,A -85,B 0,C 180,E1 -8146.628,E2 -8146.628} C_VEL
LIN {X 0,Y 460.514,Z 212.119,A -85,B 0,C 180,E1 -8149.734,E2 -8149.734} C_VEL
LIN {X 0,Y 460.475,Z 212.125,A -85,B 0,C 180,E1 -8152.527,E2 -8152.527} C_VEL
LIN {X 0,Y 460.526,Z 212.117,A -85,B 0,C 180,E1 -8155.627,E2 -8155.627} C_VEL
LIN {X 0,Y 460.518,Z 212.117,A -85,B 0,C 180,E1 -8158.748,E2 -8158.748} C_VEL
LIN {X 0,Y 460.564,Z 212.115,A -85,B 0,C 180,E1 -8162.257,E2 -8162.257} C_VEL
LIN {X 0,Y 460.525,Z 212.116,A -85,B 0,C 180,E1 -8164.708,E2 -8164.708} C_VEL
LIN {X 0,Y 460.498,Z 212.122,A -85,B 0,C 180,E1 -8167.575,E2 -8167.575} C_VEL
LIN {X 0,Y 460.557,Z 212.113,A -85,B 0,C 180,E1 -8170.387,E2 -8170.387} C_VEL
LIN {X 0,Y 460.596,Z 212.111,A -85,B 0,C 180,E1 -8174.062,E2 -8174.062} C_VEL
LIN {X 0,Y 460.603,Z 212.113,A -85,B 0,C 180,E1 -8177.668,E2 -8177.668} C_VEL
LIN {X 0,Y 460.567,Z 212.113,A -85,B 0,C 180,E1 -8179.26,E2 -8179.26} C_VEL
LIN {X 0,Y 459.907,Z 212.201,A -85,B 0,C 180,E1 -8179.99,E2 -8179.99} C_VEL
LIN {X 0,Y 457.066,Z 212.554,A -85,B 0,C 180,E1 -8181.176,E2 -8181.176} C_VEL
LIN {X 0,Y 454.673,Z 212.85,A -85,B 0,C 180,E1 -8182.133,E2 -8182.133} C_VEL
LIN {X 0,Y 453.665,Z 212.974,A -85,B 0,C 180,E1 -8182.871,E2 -8182.871} C_VEL
LIN {X 0,Y 453.593,Z 212.983,A -85,B 0,C 180,E1 -8183.122,E2 -8183.122} C_VEL
LIN {X 0,Y 453.655,Z 213.017,A -85,B 0,C 180,E1 -8184.78,E2 -8184.78} C_VEL
LIN {X 0,Y 454.596,Z 219.776,A -85,B 0,C 180,E1 -8186.235,E2 -8186.235} C_VEL
LIN {X 0,Y 454.516,Z 226.611,A -85,B 0,C 180,E1 -8187.642,E2 -8187.642} C_VEL
LIN {X 0,Y 457.598,Z 241.881,A -85,B 0,C 180,E1 -8187.999,E2 -8187.999} C_VEL
LIN {X 0,Y 456.779,Z 334.135,A -85,B 0,C 180,E1 -8189.478,E2 -8189.478} C_VEL
LIN {X 0,Y 456.452,Z 347.157,A -85,B 0,C 180,E1 -8189.864,E2 -8189.864} C_VEL
LIN {X 0,Y 456.14,Z 360.189,A -85,B 0,C 180,E1 -8190.443,E2 -8190.443} C_VEL
LIN {X 0,Y 455.694,Z 371.238,A -85,B 0,C 180,E1 -8191.106,E2 -8191.106} C_VEL
LIN {X 0,Y 455.102,Z 382.757,A -85,B 0,C 180,E1 -8191.993,E2 -8191.993} C_VEL
LIN {X 0,Y 454.571,Z 393.111,A -85,B 0,C 180,E1 -8192.992,E2 -8192.992} C_VEL
LIN {X 0,Y 454.125,Z 401.581,A -85,B 0,C 180,E1 -8193.995,E2 -8193.995} C_VEL
LIN {X 0,Y 453.757,Z 409.391,A -85,B 0,C 180,E1 -8195.111,E2 -8195.111} C_VEL
LIN {X 0,Y 453.364,Z 415.9,A -85,B 0,C 180,E1 -8196.231,E2 -8196.231} C_VEL
LIN {X 0,Y 453.101,Z 422.286,A -85,B 0,C 180,E1 -8197.577,E2 -8197.577} C_VEL
LIN {X 0,Y 452.86,Z 427.368,A -85,B 0,C 180,E1 -8198.929,E2 -8198.929} C_VEL
LIN {X 0,Y 452.684,Z 431.316,A -85,B 0,C 180,E1 -8200.285,E2 -8200.285} C_VEL
LIN {X 0,Y 452.567,Z 434.71,A -85,B 0,C 180,E1 -8201.948,E2 -8201.948} C_VEL
LIN {X 0,Y 452.422,Z 436.567,A -85,B 0,C 180,E1 -8203.475,E2 -8203.475} C_VEL
LIN {X 0,Y 452.428,Z 437.133,A -85,B 0,C 180,E1 -8204.392,E2 -8204.392} C_VEL
LIN {X 0,Y 452.441,Z 437.192,A -85,B 0,C 180,E1 -8205.619,E2 -8205.619} C_VEL
LIN {X 0,Y 452.432,Z 436.242,A -85,B 0,C 180,E1 -8207.166,E2 -8207.166} C_VEL
LIN {X 0,Y 452.579,Z 434.115,A -85,B 0,C 180,E1 -8208.693,E2 -8208.693} C_VEL
LIN {X 0,Y 452.734,Z 431.378,A -85,B 0,C 180,E1 -8209.969,E2 -8209.969} C_VEL
LIN {X 0,Y 452.923,Z 427.208,A -85,B 0,C 180,E1 -8211.407,E2 -8211.407} C_VEL
LIN {X 0,Y 453.28,Z 420.798,A -85,B 0,C 180,E1 -8213.047,E2 -8213.047} C_VEL
LIN {X 0,Y 453.683,Z 413.715,A -85,B 0,C 180,E1 -8214.461,E2 -8214.461} C_VEL
LIN {X 0,Y 454.136,Z 406.157,A -85,B 0,C 180,E1 -8215.677,E2 -8215.677} C_VEL
LIN {X 0,Y 454.689,Z 396.949,A -85,B 0,C 180,E1 -8216.878,E2 -8216.878} C_VEL
LIN {X 0,Y 455.244,Z 386.889,A -85,B 0,C 180,E1 -8217.943,E2 -8217.943} C_VEL
LIN {X 0,Y 455.927,Z 375.261,A -85,B 0,C 180,E1 -8218.922,E2 -8218.922} C_VEL
LIN {X 0,Y 456.436,Z 363.178,A -85,B 0,C 180,E1 -8219.709,E2 -8219.709} C_VEL
LIN {X 0,Y 456.873,Z 350.232,A -85,B 0,C 180,E1 -8220.339,E2 -8220.339} C_VEL
LIN {X 0,Y 457.175,Z 337.087,A -85,B 0,C 180,E1 -8220.77,E2 -8220.77} C_VEL
LIN {X 0,Y 457.386,Z 318.935,A -85,B 0,C 180,E1 -8221.107,E2 -8221.107} C_VEL
LIN {X 0,Y 458.113,Z 242.008,A -85,B 0,C 180,E1 -8222.335,E2 -8222.335} C_VEL
LIN {X 0,Y 454.825,Z 226.759,A -85,B 0,C 180,E1 -8222.738,E2 -8222.738} C_VEL
LIN {X 0,Y 454.907,Z 220.343,A -85,B 0,C 180,E1 -8224.057,E2 -8224.057} C_VEL
LIN {X 0,Y 453.492,Z 212.997,A -85,B 0,C 180,E1 -8225.667,E2 -8225.667} C_VEL
LIN {X 0,Y 453.516,Z 212.993,A -85,B 0,C 180,E1 -8229.21,E2 -8229.21} C_VEL
LIN {X 0,Y 453.485,Z 212.994,A -85,B 0,C 180,E1 -8231.936,E2 -8231.936} C_VEL
LIN {X 0,Y 453.479,Z 212.997,A -85,B 0,C 180,E1 -8235.469,E2 -8235.469} C_VEL
LIN {X 0,Y 453.476,Z 213,A -85,B 0,C 180,E1 -8238.209,E2 -8238.209} C_VEL
LIN {X 0,Y 453.508,Z 212.992,A -85,B 0,C 180,E1 -8240.787,E2 -8240.787} C_VEL
LIN {X 0,Y 453.437,Z 213.005,A -85,B 0,C 180,E1 -8243.916,E2 -8243.916} C_VEL
LIN {X 0,Y 453.462,Z 212.996,A -85,B 0,C 180,E1 -8247.15,E2 -8247.15} C_VEL
LIN {X 0,Y 453.493,Z 212.993,A -85,B 0,C 180,E1 -8250.27,E2 -8250.27} C_VEL
LIN {X 0,Y 453.482,Z 212.994,A -85,B 0,C 180,E1 -8253.293,E2 -8253.293} C_VEL
LIN {X 0,Y 453.485,Z 212.995,A -85,B 0,C 180,E1 -8256.238,E2 -8256.238} C_VEL
LIN {X 0,Y 453.482,Z 212.99,A -85,B 0,C 180,E1 -8259.118,E2 -8259.118} C_VEL
LIN {X 0,Y 453.485,Z 212.994,A -85,B 0,C 180,E1 -8261.944,E2 -8261.944} C_VEL
LIN {X 0,Y 453.522,Z 212.989,A -85,B 0,C 180,E1 -8264.726,E2 -8264.726} C_VEL
LIN {X 0,Y 453.531,Z 212.986,A -85,B 0,C 180,E1 -8268.379,E2 -8268.379} C_VEL
LIN {X 0,Y 453.624,Z 212.973,A -85,B 0,C 180,E1 -8271.985,E2 -8271.985} C_VEL
LIN {X 0,Y 453.646,Z 212.973,A -85,B 0,C 180,E1 -8274.667,E2 -8274.667} C_VEL
LIN {X 0,Y 453.713,Z 212.965,A -85,B 0,C 180,E1 -8277.337,E2 -8277.337} C_VEL
LIN {X 0,Y 453.789,Z 212.951,A -85,B 0,C 180,E1 -8280,E2 -8280} C_VEL
LIN {X 0,Y 453.712,Z 212.962,A -85,B 0,C 180,E1 -8282.664,E2 -8282.664} C_VEL
LIN {X 0,Y 453.628,Z 212.968,A -85,B 0,C 180,E1 -8286.226,E2 -8286.226} C_VEL
LIN {X 0,Y 453.558,Z 212.987,A -85,B 0,C 180,E1 -8288.914,E2 -8288.914} C_VEL
LIN {X 0,Y 453.576,Z 212.982,A -85,B 0,C 180,E1 -8292.552,E2 -8292.552} C_VEL
LIN {X 0,Y 453.518,Z 212.987,A -85,B 0,C 180,E1 -8296.197,E2 -8296.197} C_VEL
LIN {X 0,Y 453.492,Z 212.993,A -85,B 0,C 180,E1 -8299.04,E2 -8299.04} C_VEL
LIN {X 0,Y 453.45,Z 212.997,A -85,B 0,C 180,E1 -8301.838,E2 -8301.838} C_VEL
LIN {X 0,Y 453.469,Z 213.001,A -85,B 0,C 180,E1 -8304.737,E2 -8304.737} C_VEL
LIN {X 0,Y 453.468,Z 212.993,A -85,B 0,C 180,E1 -8307.951,E2 -8307.951} C_VEL
LIN {X 0,Y 453.438,Z 213.001,A -85,B 0,C 180,E1 -8310.763,E2 -8310.763} C_VEL
LIN {X 0,Y 453.447,Z 212.999,A -85,B 0,C 180,E1 -8313.916,E2 -8313.916} C_VEL
LIN {X 0,Y 453.431,Z 212.999,A -85,B 0,C 180,E1 -8317.192,E2 -8317.192} C_VEL
LIN {X 0,Y 453.48,Z 212.992,A -85,B 0,C 180,E1 -8320.611,E2 -8320.611} C_VEL
LIN {X 0,Y 453.449,Z 213.005,A -85,B 0,C 180,E1 -8324.224,E2 -8324.224} C_VEL
LIN {X 0,Y 453.437,Z 213,A -85,B 0,C 180,E1 -8327.005,E2 -8327.005} C_VEL
LIN {X 0,Y 453.462,Z 212.997,A -85,B 0,C 180,E1 -8329.414,E2 -8329.414} C_VEL
LIN {X 0,Y 453.445,Z 212.997,A -85,B 0,C 180,E1 -8332.812,E2 -8332.812} C_VEL
LIN {X 0,Y 453.472,Z 212.999,A -85,B 0,C 180,E1 -8336.089,E2 -8336.089} C_VEL
LIN {X 0,Y 453.472,Z 212.999,A -85,B 0,C 180,E1 -8339.242,E2 -8339.242} C_VEL
LIN {X 0,Y 453.506,Z 212.996,A -85,B 0,C 180,E1 -8342.297,E2 -8342.297} C_VEL
LIN {X 0,Y 453.53,Z 213.155,A -85,B 0,C 180,E1 -8342.892,E2 -8342.892} C_VEL
LIN {X 0,Y 456.115,Z 225.896,A -85,B 0,C 180,E1 -8345.381,E2 -8345.381} C_VEL
LIN {X 0,Y 456.075,Z 231.47,A -85,B 0,C 180,E1 -8346.382,E2 -8346.382} C_VEL
LIN {X 0,Y 455.052,Z 250.236,A -85,B 0,C 180,E1 -8349.666,E2 -8349.666} C_VEL
LIN {X 0,Y 454.44,Z 265.704,A -85,B 0,C 180,E1 -8352.297,E2 -8352.297} C_VEL
LIN {X 0,Y 457.824,Z 287.847,A -85,B 0,C 180,E1 -8352.807,E2 -8352.807} C_VEL
LIN {X 0,Y 457.051,Z 374.747,A -85,B 0,C 180,E1 -8354.218,E2 -8354.218} C_VEL
LIN {X 0,Y 456.579,Z 388.526,A -85,B 0,C 180,E1 -8354.63,E2 -8354.63} C_VEL
LIN {X 0,Y 455.983,Z 401.425,A -85,B 0,C 180,E1 -8355.21,E2 -8355.21} C_VEL
LIN {X 0,Y 455.408,Z 413.179,A -85,B 0,C 180,E1 -8355.933,E2 -8355.933} C_VEL
LIN {X 0,Y 454.857,Z 423.775,A -85,B 0,C 180,E1 -8356.76,E2 -8356.76} C_VEL
LIN {X 0,Y 454.318,Z 433.723,A -85,B 0,C 180,E1 -8357.719,E2 -8357.719} C_VEL
LIN {X 0,Y 453.775,Z 443.206,A -85,B 0,C 180,E1 -8358.837,E2 -8358.837} C_VEL
LIN {X 0,Y 453.256,Z 452.353,A -85,B 0,C 180,E1 -8360.179,E2 -8360.179} C_VEL
LIN {X 0,Y 452.929,Z 459.74,A -85,B 0,C 180,E1 -8361.522,E2 -8361.522} C_VEL
LIN {X 0,Y 452.671,Z 465.675,A -85,B 0,C 180,E1 -8362.864,E2 -8362.864} C_VEL
LIN {X 0,Y 452.532,Z 470.367,A -85,B 0,C 180,E1 -8364.205,E2 -8364.205} C_VEL
LIN {X 0,Y 452.487,Z 473.951,A -85,B 0,C 180,E1 -8365.545,E2 -8365.545} C_VEL
LIN {X 0,Y 452.486,Z 475.788,A -85,B 0,C 180,E1 -8366.437,E2 -8366.437} C_VEL
LIN {X 0,Y 452.523,Z 477.173,A -85,B 0,C 180,E1 -8367.328,E2 -8367.328} C_VEL
LIN {X 0,Y 452.492,Z 478.758,A -85,B 0,C 180,E1 -8369.109,E2 -8369.109} C_VEL
LIN {X 0,Y 452.471,Z 478.946,A -85,B 0,C 180,E1 -8369.998,E2 -8369.998} C_VEL
LIN {X 0,Y 452.491,Z 478.709,A -85,B 0,C 180,E1 -8370.888,E2 -8370.888} C_VEL
LIN {X 0,Y 452.522,Z 477.066,A -85,B 0,C 180,E1 -8372.669,E2 -8372.669} C_VEL
LIN {X 0,Y 452.488,Z 475.624,A -85,B 0,C 180,E1 -8373.56,E2 -8373.56} C_VEL
LIN {X 0,Y 452.548,Z 472.635,A -85,B 0,C 180,E1 -8374.898,E2 -8374.898} C_VEL
LIN {X 0,Y 452.609,Z 468.022,A -85,B 0,C 180,E1 -8376.394,E2 -8376.394} C_VEL
LIN {X 0,Y 452.822,Z 461.33,A -85,B 0,C 180,E1 -8378.027,E2 -8378.027} C_VEL
LIN {X 0,Y 453.085,Z 454.291,A -85,B 0,C 180,E1 -8379.371,E2 -8379.371} C_VEL
LIN {X 0,Y 453.484,Z 445.467,A -85,B 0,C 180,E1 -8380.715,E2 -8380.715} C_VEL
LIN {X 0,Y 454.057,Z 435.45,A -85,B 0,C 180,E1 -8381.945,E2 -8381.945} C_VEL
LIN {X 0,Y 454.571,Z 424.615,A -85,B 0,C 180,E1 -8383.006,E2 -8383.006} C_VEL
LIN {X 0,Y 455.116,Z 413.899,A -85,B 0,C 180,E1 -8383.846,E2 -8383.846} C_VEL
LIN {X 0,Y 455.634,Z 402.149,A -85,B 0,C 180,E1 -8384.57,E2 -8384.57} C_VEL
LIN {X 0,Y 456.138,Z 389.365,A -85,B 0,C 180,E1 -8385.153,E2 -8385.153} C_VEL
LIN {X 0,Y 456.578,Z 375.749,A -85,B 0,C 180,E1 -8385.567,E2 -8385.567} C_VEL
LIN {X 0,Y 456.917,Z 344.421,A -85,B 0,C 180,E1 -8386.09,E2 -8386.09} C_VEL
LIN {X 0,Y 457.215,Z 286.406,A -85,B 0,C 180,E1 -8387.01,E2 -8387.01} C_VEL
LIN {X 0,Y 454.222,Z 265.76,A -85,B 0,C 180,E1 -8387.453,E2 -8387.453} C_VEL
LIN {X 0,Y 454.854,Z 248.878,A -85,B 0,C 180,E1 -8390.34,E2 -8390.34} C_VEL
LIN {X 0,Y 455.749,Z 231.17,A -85,B 0,C 180,E1 -8393.392,E2 -8393.392} C_VEL
LIN {X 0,Y 455.774,Z 224.719,A -85,B 0,C 180,E1 -8394.525,E2 -8394.525} C_VEL
LIN {X 0,Y 453.592,Z 212.986,A -85,B 0,C 180,E1 -8396.758,E2 -8396.758} C_VEL
LIN {X 0,Y 453.458,Z 213.003,A -85,B 0,C 180,E1 -8399.781,E2 -8399.781} C_VEL
LIN {X 0,Y 453.474,Z 212.994,A -85,B 0,C 180,E1 -8403.185,E2 -8403.185} C_VEL
LIN {X 0,Y 453.435,Z 213.003,A -85,B 0,C 180,E1 -8406.295,E2 -8406.295} C_VEL
LIN {X 0,Y 453.466,Z 212.997,A -85,B 0,C 180,E1 -8409.446,E2 -8409.446} C_VEL
LIN {X 0,Y 453.451,Z 213.004,A -85,B 0,C 180,E1 -8411.931,E2 -8411.931} C_VEL
LIN {X 0,Y 453.464,Z 212.998,A -85,B 0,C 180,E1 -8415.466,E2 -8415.466} C_VEL
LIN {X 0,Y 453.466,Z 212.998,A -85,B 0,C 180,E1 -8418.207,E2 -8418.207} C_VEL
LIN {X 0,Y 453.502,Z 212.99,A -85,B 0,C 180,E1 -8420.783,E2 -8420.783} C_VEL
LIN {X 0,Y 453.42,Z 213.005,A -85,B 0,C 180,E1 -8423.914,E2 -8423.914} C_VEL
LIN {X 0,Y 453.444,Z 213,A -85,B 0,C 180,E1 -8427.148,E2 -8427.148} C_VEL
LIN {X 0,Y 453.474,Z 212.995,A -85,B 0,C 180,E1 -8430.268,E2 -8430.268} C_VEL
LIN {X 0,Y 453.469,Z 212.999,A -85,B 0,C 180,E1 -8433.291,E2 -8433.291} C_VEL
LIN {X 0,Y 453.471,Z 212.995,A -85,B 0,C 180,E1 -8436.237,E2 -8436.237} C_VEL
LIN {X 0,Y 453.471,Z 212.998,A -85,B 0,C 180,E1 -8439.117,E2 -8439.117} C_VEL
LIN {X 0,Y 453.464,Z 212.997,A -85,B 0,C 180,E1 -8441.942,E2 -8441.942} C_VEL
LIN {X 0,Y 453.501,Z 212.992,A -85,B 0,C 180,E1 -8444.725,E2 -8444.725} C_VEL
LIN {X 0,Y 453.538,Z 212.986,A -85,B 0,C 180,E1 -8448.378,E2 -8448.378} C_VEL
LIN {X 0,Y 453.606,Z 212.978,A -85,B 0,C 180,E1 -8451.984,E2 -8451.984} C_VEL
LIN {X 0,Y 453.628,Z 212.977,A -85,B 0,C 180,E1 -8454.666,E2 -8454.666} C_VEL
LIN {X 0,Y 453.712,Z 212.969,A -85,B 0,C 180,E1 -8457.336,E2 -8457.336} C_VEL
LIN {X 0,Y 453.767,Z 212.957,A -85,B 0,C 180,E1 -8460,E2 -8460} C_VEL
LIN {X 0,Y 453.691,Z 212.97,A -85,B 0,C 180,E1 -8462.663,E2 -8462.663} C_VEL
LIN {X 0,Y 453.616,Z 212.977,A -85,B 0,C 180,E1 -8466.226,E2 -8466.226} C_VEL
LIN {X 0,Y 453.541,Z 212.994,A -85,B 0,C 180,E1 -8468.914,E2 -8468.914} C_VEL
LIN {X 0,Y 453.551,Z 212.988,A -85,B 0,C 180,E1 -8472.552,E2 -8472.552} C_VEL
LIN {X 0,Y 453.506,Z 212.991,A -85,B 0,C 180,E1 -8476.197,E2 -8476.197} C_VEL
LIN {X 0,Y 453.469,Z 212.999,A -85,B 0,C 180,E1 -8479.042,E2 -8479.042} C_VEL
LIN {X 0,Y 453.43,Z 212.999,A -85,B 0,C 180,E1 -8481.838,E2 -8481.838} C_VEL
LIN {X 0,Y 453.468,Z 213.002,A -85,B 0,C 180,E1 -8484.737,E2 -8484.737} C_VEL
LIN {X 0,Y 453.487,Z 212.993,A -85,B 0,C 180,E1 -8487.962,E2 -8487.962} C_VEL
LIN {X 0,Y 453.423,Z 213,A -85,B 0,C 180,E1 -8491.528,E2 -8491.528} C_VEL
LIN {X 0,Y 453.449,Z 213.001,A -85,B 0,C 180,E1 -8494.78,E2 -8494.78} C_VEL
LIN {X 0,Y 453.423,Z 213.007,A -85,B 0,C 180,E1 -8498.315,E2 -8498.315} C_VEL
LIN {X 0,Y 453.459,Z 213.001,A -85,B 0,C 180,E1 -8500.612,E2 -8500.612} C_VEL
LIN {X 0,Y 453.419,Z 213.001,A -85,B 0,C 180,E1 -8503.247,E2 -8503.247} C_VEL
LIN {X 0,Y 453.43,Z 213.001,A -85,B 0,C 180,E1 -8505.782,E2 -8505.782} C_VEL
LIN {X 0,Y 453.451,Z 213.004,A -85,B 0,C 180,E1 -8508.213,E2 -8508.213} C_VEL
LIN {X 0,Y 453.488,Z 212.993,A -85,B 0,C 180,E1 -8510.794,E2 -8510.794} C_VEL
LIN {X 0,Y 453.432,Z 213.004,A -85,B 0,C 180,E1 -8513.921,E2 -8513.921} C_VEL
LIN {X 0,Y 453.462,Z 212.995,A -85,B 0,C 180,E1 -8517.155,E2 -8517.155} C_VEL
LIN {X 0,Y 453.456,Z 213.001,A -85,B 0,C 180,E1 -8520.272,E2 -8520.272} C_VEL
LIN {X 0,Y 453.486,Z 212.993,A -85,B 0,C 180,E1 -8523.297,E2 -8523.297} C_VEL
LIN {X 0,Y 453.484,Z 212.997,A -85,B 0,C 180,E1 -8526.242,E2 -8526.242} C_VEL
LIN {X 0,Y 453.47,Z 212.995,A -85,B 0,C 180,E1 -8529.121,E2 -8529.121} C_VEL
LIN {X 0,Y 453.492,Z 212.998,A -85,B 0,C 180,E1 -8531.947,E2 -8531.947} C_VEL
LIN {X 0,Y 453.53,Z 212.987,A -85,B 0,C 180,E1 -8534.729,E2 -8534.729} C_VEL
LIN {X 0,Y 453.553,Z 212.985,A -85,B 0,C 180,E1 -8538.381,E2 -8538.381} C_VEL
LIN {X 0,Y 453.581,Z 212.982,A -85,B 0,C 180,E1 -8541.089,E2 -8541.089} C_VEL
LIN {X 0,Y 453.593,Z 212.983,A -85,B 0,C 180,E1 -8543.122,E2 -8543.122} C_VEL
LIN {X 0,Y 452.969,Z 213.188,A -85,B 0,C 180,E1 -8543.624,E2 -8543.624} C_VEL
LIN {X 0,Y 450.32,Z 214.358,A -85,B 0,C 180,E1 -8544.407,E2 -8544.407} C_VEL
LIN {X 0,Y 447.77,Z 216.578,A -85,B 0,C 180,E1 -8545.162,E2 -8545.162} C_VEL
LIN {X 0,Y 447.306,Z 218.448,A -85,B 0,C 180,E1 -8545.615,E2 -8545.615} C_VEL
LIN {X 0,Y 447.62,Z 223.194,A -85,B 0,C 180,E1 -8546.626,E2 -8546.626} C_VEL
LIN {X 0,Y 447.574,Z 227.098,A -85,B 0,C 180,E1 -8547.399,E2 -8547.399} C_VEL
LIN {X 0,Y 450.805,Z 243.427,A -85,B 0,C 180,E1 -8547.785,E2 -8547.785} C_VEL
LIN {X 0,Y 449.917,Z 333.819,A -85,B 0,C 180,E1 -8549.249,E2 -8549.249} C_VEL
LIN {X 0,Y 449.593,Z 346.955,A -85,B 0,C 180,E1 -8549.637,E2 -8549.637} C_VEL
LIN {X 0,Y 449.259,Z 359.044,A -85,B 0,C 180,E1 -8550.17,E2 -8550.17} C_VEL
LIN {X 0,Y 448.805,Z 371.286,A -85,B 0,C 180,E1 -8550.899,E2 -8550.899} C_VEL
LIN {X 0,Y 448.155,Z 382.868,A -85,B 0,C 180,E1 -8551.799,E2 -8551.799} C_VEL
LIN {X 0,Y 447.591,Z 393.265,A -85,B 0,C 180,E1 -8552.814,E2 -8552.814} C_VEL
LIN {X 0,Y 447.137,Z 401.767,A -85,B 0,C 180,E1 -8553.831,E2 -8553.831} C_VEL
LIN {X 0,Y 446.723,Z 409.615,A -85,B 0,C 180,E1 -8554.965,E2 -8554.965} C_VEL
LIN {X 0,Y 446.294,Z 417.295,A -85,B 0,C 180,E1 -8556.33,E2 -8556.33} C_VEL
LIN {X 0,Y 446.004,Z 423.461,A -85,B 0,C 180,E1 -8557.698,E2 -8557.698} C_VEL
LIN {X 0,Y 445.757,Z 428.368,A -85,B 0,C 180,E1 -8559.072,E2 -8559.072} C_VEL
LIN {X 0,Y 445.602,Z 432.148,A -85,B 0,C 180,E1 -8560.451,E2 -8560.451} C_VEL
LIN {X 0,Y 445.476,Z 435.167,A -85,B 0,C 180,E1 -8562.005,E2 -8562.005} C_VEL
LIN {X 0,Y 445.349,Z 437.08,A -85,B 0,C 180,E1 -8563.693,E2 -8563.693} C_VEL
LIN {X 0,Y 445.343,Z 437.508,A -85,B 0,C 180,E1 -8564.626,E2 -8564.626} C_VEL
LIN {X 0,Y 445.342,Z 437.511,A -85,B 0,C 180,E1 -8565.71,E2 -8565.71} C_VEL
LIN {X 0,Y 445.358,Z 436.336,A -85,B 0,C 180,E1 -8567.447,E2 -8567.447} C_VEL
LIN {X 0,Y 445.509,Z 434.355,A -85,B 0,C 180,E1 -8568.825,E2 -8568.825} C_VEL
LIN {X 0,Y 445.678,Z 431.142,A -85,B 0,C 180,E1 -8570.299,E2 -8570.299} C_VEL
LIN {X 0,Y 445.927,Z 426.464,A -85,B 0,C 180,E1 -8571.845,E2 -8571.845} C_VEL
LIN {X 0,Y 446.331,Z 420.219,A -85,B 0,C 180,E1 -8573.41,E2 -8573.41} C_VEL
LIN {X 0,Y 446.707,Z 414.042,A -85,B 0,C 180,E1 -8574.64,E2 -8574.64} C_VEL
LIN {X 0,Y 447.201,Z 406.612,A -85,B 0,C 180,E1 -8575.855,E2 -8575.855} C_VEL
LIN {X 0,Y 447.777,Z 397.435,A -85,B 0,C 180,E1 -8577.075,E2 -8577.075} C_VEL
LIN {X 0,Y 448.297,Z 388.451,A -85,B 0,C 180,E1 -8578.054,E2 -8578.054} C_VEL
LIN {X 0,Y 448.986,Z 377.389,A -85,B 0,C 180,E1 -8579.027,E2 -8579.027} C_VEL
LIN {X 0,Y 449.536,Z 365.952,A -85,B 0,C 180,E1 -8579.824,E2 -8579.824} C_VEL
LIN {X 0,Y 450.021,Z 353.805,A -85,B 0,C 180,E1 -8580.461,E2 -8580.461} C_VEL
LIN {X 0,Y 450.364,Z 340.427,A -85,B 0,C 180,E1 -8580.959,E2 -8580.959} C_VEL
LIN {X 0,Y 450.548,Z 327.132,A -85,B 0,C 180,E1 -8581.257,E2 -8581.257} C_VEL
LIN {X 0,Y 451.519,Z 244.089,A -85,B 0,C 180,E1 -8582.599,E2 -8582.599} C_VEL
LIN {X 0,Y 448.373,Z 228.919,A -85,B 0,C 180,E1 -8583.002,E2 -8583.002} C_VEL
LIN {X 0,Y 447.962,Z 226.941,A -85,B 0,C 180,E1 -8583.084,E2 -8583.084} C_VEL
LIN {X 0,Y 447.863,Z 220.692,A -85,B 0,C 180,E1 -8584.395,E2 -8584.395} C_VEL
LIN {X 0,Y 446.439,Z 213.876,A -85,B 0,C 180,E1 -8585.935,E2 -8585.935} C_VEL
LIN {X 0,Y 446.478,Z 213.87,A -85,B 0,C 180,E1 -8589.529,E2 -8589.529} C_VEL
LIN {X 0,Y 446.438,Z 213.879,A -85,B 0,C 180,E1 -8592.601,E2 -8592.601} C_VEL
LIN {X 0,Y 446.444,Z 213.873,A -85,B 0,C 180,E1 -8595.102,E2 -8595.102} C_VEL
LIN {X 0,Y 446.426,Z 213.876,A -85,B 0,C 180,E1 -8598.609,E2 -8598.609} C_VEL
LIN {X 0,Y 446.452,Z 213.871,A -85,B 0,C 180,E1 -8600.974,E2 -8600.974} C_VEL
LIN {X 0,Y 446.402,Z 213.877,A -85,B 0,C 180,E1 -8604.373,E2 -8604.373} C_VEL
LIN {X 0,Y 446.402,Z 213.879,A -85,B 0,C 180,E1 -8607.637,E2 -8607.637} C_VEL
LIN {X 0,Y 446.447,Z 213.868,A -85,B 0,C 180,E1 -8610.791,E2 -8610.791} C_VEL
LIN {X 0,Y 446.455,Z 213.872,A -85,B 0,C 180,E1 -8613.847,E2 -8613.847} C_VEL
LIN {X 0,Y 446.416,Z 213.873,A -85,B 0,C 180,E1 -8616.823,E2 -8616.823} C_VEL
LIN {X 0,Y 446.431,Z 213.874,A -85,B 0,C 180,E1 -8619.737,E2 -8619.737} C_VEL
LIN {X 0,Y 446.439,Z 213.867,A -85,B 0,C 180,E1 -8622.596,E2 -8622.596} C_VEL
LIN {X 0,Y 446.446,Z 213.876,A -85,B 0,C 180,E1 -8625.412,E2 -8625.412} C_VEL
LIN {X 0,Y 446.489,Z 213.864,A -85,B 0,C 180,E1 -8628.193,E2 -8628.193} C_VEL
LIN {X 0,Y 446.572,Z 213.852,A -85,B 0,C 180,E1 -8631.858,E2 -8631.858} C_VEL
LIN {X 0,Y 446.621,Z 213.847,A -85,B 0,C 180,E1 -8634.583,E2 -8634.583} C_VEL
LIN {X 0,Y 446.632,Z 213.844,A -85,B 0,C 180,E1 -8638.197,E2 -8638.197} C_VEL
LIN {X 0,Y 446.76,Z 213.827,A -85,B 0,C 180,E1 -8640,E2 -8640} C_VEL
LIN {X 0,Y 446.659,Z 213.841,A -85,B 0,C 180,E1 -8642.706,E2 -8642.706} C_VEL
LIN {X 0,Y 446.596,Z 213.844,A -85,B 0,C 180,E1 -8646.325,E2 -8646.325} C_VEL
LIN {X 0,Y 446.506,Z 213.863,A -85,B 0,C 180,E1 -8649.056,E2 -8649.056} C_VEL
LIN {X 0,Y 446.507,Z 213.864,A -85,B 0,C 180,E1 -8652.73,E2 -8652.73} C_VEL
LIN {X 0,Y 446.463,Z 213.868,A -85,B 0,C 180,E1 -8656.46,E2 -8656.46} C_VEL
LIN {X 0,Y 446.443,Z 213.87,A -85,B 0,C 180,E1 -8659.305,E2 -8659.305} C_VEL
LIN {X 0,Y 446.391,Z 213.878,A -85,B 0,C 180,E1 -8662.201,E2 -8662.201} C_VEL
LIN {X 0,Y 446.414,Z 213.877,A -85,B 0,C 180,E1 -8665.155,E2 -8665.155} C_VEL
LIN {X 0,Y 446.42,Z 213.873,A -85,B 0,C 180,E1 -8668.183,E2 -8668.183} C_VEL
LIN {X 0,Y 446.388,Z 213.876,A -85,B 0,C 180,E1 -8671.303,E2 -8671.303} C_VEL
LIN {X 0,Y 446.403,Z 213.878,A -85,B 0,C 180,E1 -8674.526,E2 -8674.526} C_VEL
LIN {X 0,Y 446.393,Z 213.878,A -85,B 0,C 180,E1 -8678.08,E2 -8678.08} C_VEL
LIN {X 0,Y 446.405,Z 213.868,A -85,B 0,C 180,E1 -8681.394,E2 -8681.394} C_VEL
LIN {X 0,Y 446.411,Z 213.876,A -85,B 0,C 180,E1 -8684.894,E2 -8684.894} C_VEL
LIN {X 0,Y 446.41,Z 213.877,A -85,B 0,C 180,E1 -8687.727,E2 -8687.727} C_VEL
LIN {X 0,Y 446.4,Z 213.877,A -85,B 0,C 180,E1 -8690.971,E2 -8690.971} C_VEL
LIN {X 0,Y 446.414,Z 213.88,A -85,B 0,C 180,E1 -8694.375,E2 -8694.375} C_VEL
LIN {X 0,Y 446.418,Z 213.878,A -85,B 0,C 180,E1 -8697.64,E2 -8697.64} C_VEL
LIN {X 0,Y 446.435,Z 213.875,A -85,B 0,C 180,E1 -8700.791,E2 -8700.791} C_VEL
LIN {X 0,Y 446.482,Z 213.904,A -85,B 0,C 180,E1 -8702.587,E2 -8702.587} C_VEL
LIN {X 0,Y 449.149,Z 226.858,A -85,B 0,C 180,E1 -8705.169,E2 -8705.169} C_VEL
LIN {X 0,Y 449.264,Z 231.349,A -85,B 0,C 180,E1 -8706.001,E2 -8706.001} C_VEL
LIN {X 0,Y 448.161,Z 250.109,A -85,B 0,C 180,E1 -8709.339,E2 -8709.339} C_VEL
LIN {X 0,Y 447.491,Z 265.172,A -85,B 0,C 180,E1 -8711.973,E2 -8711.973} C_VEL
LIN {X 0,Y 451.089,Z 288.272,A -85,B 0,C 180,E1 -8712.524,E2 -8712.524} C_VEL
LIN {X 0,Y 450.292,Z 374.44,A -85,B 0,C 180,E1 -8713.946,E2 -8713.946} C_VEL
LIN {X 0,Y 449.807,Z 388.207,A -85,B 0,C 180,E1 -8714.364,E2 -8714.364} C_VEL
LIN {X 0,Y 449.194,Z 400.589,A -85,B 0,C 180,E1 -8714.923,E2 -8714.923} C_VEL
LIN {X 0,Y 448.608,Z 411.668,A -85,B 0,C 180,E1 -8715.599,E2 -8715.599} C_VEL
LIN {X 0,Y 447.965,Z 423.486,A -85,B 0,C 180,E1 -8716.527,E2 -8716.527} C_VEL
LIN {X 0,Y 447.351,Z 433.661,A -85,B 0,C 180,E1 -8717.524,E2 -8717.524} C_VEL
LIN {X 0,Y 446.797,Z 443.073,A -85,B 0,C 180,E1 -8718.66,E2 -8718.66} C_VEL
LIN {X 0,Y 446.223,Z 452.171,A -85,B 0,C 180,E1 -8720.023,E2 -8720.023} C_VEL
LIN {X 0,Y 445.865,Z 459.523,A -85,B 0,C 180,E1 -8721.387,E2 -8721.387} C_VEL
LIN {X 0,Y 445.599,Z 465.432,A -85,B 0,C 180,E1 -8722.75,E2 -8722.75} C_VEL
LIN {X 0,Y 445.446,Z 469.697,A -85,B 0,C 180,E1 -8723.985,E2 -8723.985} C_VEL
LIN {X 0,Y 445.413,Z 473.672,A -85,B 0,C 180,E1 -8725.474,E2 -8725.474} C_VEL
LIN {X 0,Y 445.385,Z 475.493,A -85,B 0,C 180,E1 -8726.38,E2 -8726.38} C_VEL
LIN {X 0,Y 445.447,Z 476.872,A -85,B 0,C 180,E1 -8727.286,E2 -8727.286} C_VEL
LIN {X 0,Y 445.398,Z 478.442,A -85,B 0,C 180,E1 -8729.094,E2 -8729.094} C_VEL
LIN {X 0,Y 445.407,Z 478.616,A -85,B 0,C 180,E1 -8729.998,E2 -8729.998} C_VEL
LIN {X 0,Y 445.399,Z 477.736,A -85,B 0,C 180,E1 -8731.807,E2 -8731.807} C_VEL
LIN {X 0,Y 445.446,Z 476.712,A -85,B 0,C 180,E1 -8732.711,E2 -8732.711} C_VEL
LIN {X 0,Y 445.389,Z 475.253,A -85,B 0,C 180,E1 -8733.617,E2 -8733.617} C_VEL
LIN {X 0,Y 445.477,Z 472.251,A -85,B 0,C 180,E1 -8734.976,E2 -8734.976} C_VEL
LIN {X 0,Y 445.549,Z 466.715,A -85,B 0,C 180,E1 -8736.746,E2 -8736.746} C_VEL
LIN {X 0,Y 445.749,Z 460.901,A -85,B 0,C 180,E1 -8738.155,E2 -8738.155} C_VEL
LIN {X 0,Y 446.034,Z 453.83,A -85,B 0,C 180,E1 -8739.521,E2 -8739.521} C_VEL
LIN {X 0,Y 446.483,Z 444.969,A -85,B 0,C 180,E1 -8740.885,E2 -8740.885} C_VEL
LIN {X 0,Y 446.997,Z 434.897,A -85,B 0,C 180,E1 -8742.137,E2 -8742.137} C_VEL
LIN {X 0,Y 447.623,Z 423.75,A -85,B 0,C 180,E1 -8743.232,E2 -8743.232} C_VEL
LIN {X 0,Y 448.162,Z 413.184,A -85,B 0,C 180,E1 -8744.065,E2 -8744.065} C_VEL
LIN {X 0,Y 448.739,Z 401.322,A -85,B 0,C 180,E1 -8744.799,E2 -8744.799} C_VEL
LIN {X 0,Y 449.227,Z 388.246,A -85,B 0,C 180,E1 -8745.392,E2 -8745.392} C_VEL
LIN {X 0,Y 449.674,Z 375.367,A -85,B 0,C 180,E1 -8745.783,E2 -8745.783} C_VEL
LIN {X 0,Y 450.008,Z 348.769,A -85,B 0,C 180,E1 -8746.236,E2 -8746.236} C_VEL
LIN {X 0,Y 450.448,Z 287.728,A -85,B 0,C 180,E1 -8747.216,E2 -8747.216} C_VEL
LIN {X 0,Y 447.252,Z 265.429,A -85,B 0,C 180,E1 -8747.705,E2 -8747.705} C_VEL
LIN {X 0,Y 447.997,Z 247.002,A -85,B 0,C 180,E1 -8750.906,E2 -8750.906} C_VEL
LIN {X 0,Y 448.83,Z 230.622,A -85,B 0,C 180,E1 -8753.775,E2 -8753.775} C_VEL
LIN {X 0,Y 448.96,Z 227.342,A -85,B 0,C 180,E1 -8754.355,E2 -8754.355} C_VEL
LIN {X 0,Y 446.765,Z 214.988,A -85,B 0,C 180,E1 -8756.689,E2 -8756.689} C_VEL
LIN {X 0,Y 446.542,Z 213.864,A -85,B 0,C 180,E1 -8756.927,E2 -8756.927} C_VEL
LIN {X 0,Y 446.413,Z 213.879,A -85,B 0,C 180,E1 -8760.246,E2 -8760.246} C_VEL
LIN {X 0,Y 446.428,Z 213.873,A -85,B 0,C 180,E1 -8763.45,E2 -8763.45} C_VEL
LIN {X 0,Y 446.382,Z 213.878,A -85,B 0,C 180,E1 -8766.741,E2 -8766.741} C_VEL
LIN {X 0,Y 446.42,Z 213.877,A -85,B 0,C 180,E1 -8770.194,E2 -8770.194} C_VEL
LIN {X 0,Y 446.403,Z 213.875,A -85,B 0,C 180,E1 -8772.601,E2 -8772.601} C_VEL
LIN {X 0,Y 446.428,Z 213.872,A -85,B 0,C 180,E1 -8775.099,E2 -8775.099} C_VEL
LIN {X 0,Y 446.414,Z 213.874,A -85,B 0,C 180,E1 -8778.607,E2 -8778.607} C_VEL
LIN {X 0,Y 446.444,Z 213.87,A -85,B 0,C 180,E1 -8780.973,E2 -8780.973} C_VEL
LIN {X 0,Y 446.385,Z 213.878,A -85,B 0,C 180,E1 -8784.37,E2 -8784.37} C_VEL
LIN {X 0,Y 446.384,Z 213.885,A -85,B 0,C 180,E1 -8787.635,E2 -8787.635} C_VEL
LIN {X 0,Y 446.429,Z 213.872,A -85,B 0,C 180,E1 -8790.789,E2 -8790.789} C_VEL
LIN {X 0,Y 446.435,Z 213.874,A -85,B 0,C 180,E1 -8793.845,E2 -8793.845} C_VEL
LIN {X 0,Y 446.401,Z 213.876,A -85,B 0,C 180,E1 -8796.822,E2 -8796.822} C_VEL
LIN {X 0,Y 446.413,Z 213.877,A -85,B 0,C 180,E1 -8799.735,E2 -8799.735} C_VEL
LIN {X 0,Y 446.417,Z 213.873,A -85,B 0,C 180,E1 -8802.595,E2 -8802.595} C_VEL
LIN {X 0,Y 446.428,Z 213.878,A -85,B 0,C 180,E1 -8805.411,E2 -8805.411} C_VEL
LIN {X 0,Y 446.497,Z 213.863,A -85,B 0,C 180,E1 -8808.192,E2 -8808.192} C_VEL
LIN {X 0,Y 446.555,Z 213.857,A -85,B 0,C 180,E1 -8811.857,E2 -8811.857} C_VEL
LIN {X 0,Y 446.602,Z 213.851,A -85,B 0,C 180,E1 -8814.582,E2 -8814.582} C_VEL
LIN {X 0,Y 446.656,Z 213.849,A -85,B 0,C 180,E1 -8817.294,E2 -8817.294} C_VEL
LIN {X 0,Y 446.738,Z 213.833,A -85,B 0,C 180,E1 -8820,E2 -8820} C_VEL
LIN {X 0,Y 446.638,Z 213.849,A -85,B 0,C 180,E1 -8822.705,E2 -8822.705} C_VEL
LIN {X 0,Y 446.585,Z 213.853,A -85,B 0,C 180,E1 -8826.324,E2 -8826.324} C_VEL
LIN {X 0,Y 446.487,Z 213.87,A -85,B 0,C 180,E1 -8829.056,E2 -8829.056} C_VEL
LIN {X 0,Y 446.483,Z 213.871,A -85,B 0,C 180,E1 -8832.731,E2 -8832.731} C_VEL
LIN {X 0,Y 446.446,Z 213.873,A -85,B 0,C 180,E1 -8836.46,E2 -8836.46} C_VEL
LIN {X 0,Y 446.42,Z 213.874,A -85,B 0,C 180,E1 -8839.305,E2 -8839.305} C_VEL
LIN {X 0,Y 446.372,Z 213.881,A -85,B 0,C 180,E1 -8842.202,E2 -8842.202} C_VEL
LIN {X 0,Y 446.411,Z 213.876,A -85,B 0,C 180,E1 -8845.155,E2 -8845.155} C_VEL
LIN {X 0,Y 446.442,Z 213.873,A -85,B 0,C 180,E1 -8848.181,E2 -8848.181} C_VEL
LIN {X 0,Y 446.376,Z 213.878,A -85,B 0,C 180,E1 -8851.777,E2 -8851.777} C_VEL
LIN {X 0,Y 446.391,Z 213.884,A -85,B 0,C 180,E1 -8854.526,E2 -8854.526} C_VEL
LIN {X 0,Y 446.376,Z 213.882,A -85,B 0,C 180,E1 -8858.082,E2 -8858.082} C_VEL
LIN {X 0,Y 446.394,Z 213.876,A -85,B 0,C 180,E1 -8861.395,E2 -8861.395} C_VEL
LIN {X 0,Y 446.419,Z 213.873,A -85,B 0,C 180,E1 -8865.108,E2 -8865.108} C_VEL
LIN {X 0,Y 446.4,Z 213.878,A -85,B 0,C 180,E1 -8868.613,E2 -8868.613} C_VEL
LIN {X 0,Y 446.433,Z 213.871,A -85,B 0,C 180,E1 -8870.978,E2 -8870.978} C_VEL
LIN {X 0,Y 446.398,Z 213.88,A -85,B 0,C 180,E1 -8874.378,E2 -8874.378} C_VEL
LIN {X 0,Y 446.402,Z 213.877,A -85,B 0,C 180,E1 -8877.642,E2 -8877.642} C_VEL
LIN {X 0,Y 446.43,Z 213.872,A -85,B 0,C 180,E1 -8880.794,E2 -8880.794} C_VEL
LIN {X 0,Y 446.463,Z 213.873,A -85,B 0,C 180,E1 -8883.852,E2 -8883.852} C_VEL
LIN {X 0,Y 446.413,Z 213.873,A -85,B 0,C 180,E1 -8886.826,E2 -8886.826} C_VEL
LIN {X 0,Y 446.432,Z 213.877,A -85,B 0,C 180,E1 -8889.74,E2 -8889.74} C_VEL
LIN {X 0,Y 446.445,Z 213.87,A -85,B 0,C 180,E1 -8892.6,E2 -8892.6} C_VEL
LIN {X 0,Y 446.459,Z 213.871,A -85,B 0,C 180,E1 -8895.415,E2 -8895.415} C_VEL
LIN {X 0,Y 446.511,Z 213.864,A -85,B 0,C 180,E1 -8898.196,E2 -8898.196} C_VEL
LIN {X 0,Y 446.528,Z 213.86,A -85,B 0,C 180,E1 -8900.947,E2 -8900.947} C_VEL
LIN {X 0,Y 446.616,Z 213.856,A -85,B 0,C 180,E1 -8903.678,E2 -8903.678} C_VEL
LIN {X 0,Y 446.633,Z 213.984,A -85,B 0,C 180,E1 -8904.641,E2 -8904.641} C_VEL
LIN {X 0,Y 447.306,Z 218.448,A -85,B 0,C 180,E1 -8905.615,E2 -8905.615} C_VEL
LIN {X 0,Y 446.829,Z 220.743,A -85,B 0,C 180,E1 -8906.059,E2 -8906.059} C_VEL
LIN {X 0,Y 445.433,Z 223.295,A -85,B 0,C 180,E1 -8906.456,E2 -8906.456} C_VEL
LIN {X 0,Y 443.264,Z 227.148,A -85,B 0,C 180,E1 -8906.899,E2 -8906.899} C_VEL
LIN {X 0,Y 442.098,Z 230.529,A -85,B 0,C 180,E1 -8907.154,E2 -8907.154} C_VEL
LIN {X 0,Y 441.961,Z 233.987,A -85,B 0,C 180,E1 -8907.307,E2 -8907.307} C_VEL
LIN {X 0,Y 442.015,Z 234.31,A -85,B 0,C 180,E1 -8907.315,E2 -8907.315} C_VEL
LIN {X 0,Y 443.978,Z 245.044,A -85,B 0,C 180,E1 -8907.565,E2 -8907.565} C_VEL
LIN {X 0,Y 443.035,Z 334.773,A -85,B 0,C 180,E1 -8909.045,E2 -8909.045} C_VEL
LIN {X 0,Y 442.679,Z 348.058,A -85,B 0,C 180,E1 -8909.453,E2 -8909.453} C_VEL
LIN {X 0,Y 442.34,Z 360.106,A -85,B 0,C 180,E1 -8910.002,E2 -8910.002} C_VEL
LIN {X 0,Y 441.9,Z 371.338,A -85,B 0,C 180,E1 -8910.685,E2 -8910.685} C_VEL
LIN {X 0,Y 441.233,Z 382.972,A -85,B 0,C 180,E1 -8911.599,E2 -8911.599} C_VEL
LIN {X 0,Y 440.629,Z 393.411,A -85,B 0,C 180,E1 -8912.63,E2 -8912.63} C_VEL
LIN {X 0,Y 440.165,Z 401.939,A -85,B 0,C 180,E1 -8913.663,E2 -8913.663} C_VEL
LIN {X 0,Y 439.692,Z 409.821,A -85,B 0,C 180,E1 -8914.815,E2 -8914.815} C_VEL
LIN {X 0,Y 439.242,Z 417.531,A -85,B 0,C 180,E1 -8916.201,E2 -8916.201} C_VEL
LIN {X 0,Y 439.011,Z 422.797,A -85,B 0,C 180,E1 -8917.359,E2 -8917.359} C_VEL
LIN {X 0,Y 438.739,Z 427.915,A -85,B 0,C 180,E1 -8918.754,E2 -8918.754} C_VEL
LIN {X 0,Y 438.521,Z 431.893,A -85,B 0,C 180,E1 -8920.155,E2 -8920.155} C_VEL
LIN {X 0,Y 438.443,Z 433.936,A -85,B 0,C 180,E1 -8921.091,E2 -8921.091} C_VEL
LIN {X 0,Y 438.388,Z 435.616,A -85,B 0,C 180,E1 -8922.064,E2 -8922.064} C_VEL
LIN {X 0,Y 438.279,Z 436.777,A -85,B 0,C 180,E1 -8922.974,E2 -8922.974} C_VEL
LIN {X 0,Y 438.245,Z 437.527,A -85,B 0,C 180,E1 -8923.919,E2 -8923.919} C_VEL
LIN {X 0,Y 438.271,Z 437.875,A -85,B 0,C 180,E1 -8924.867,E2 -8924.867} C_VEL
LIN {X 0,Y 438.242,Z 437.828,A -85,B 0,C 180,E1 -8925.821,E2 -8925.821} C_VEL
LIN {X 0,Y 438.231,Z 437.336,A -85,B 0,C 180,E1 -8926.778,E2 -8926.778} C_VEL
LIN {X 0,Y 438.29,Z 436.399,A -85,B 0,C 180,E1 -8927.738,E2 -8927.738} C_VEL
LIN {X 0,Y 438.452,Z 434.59,A -85,B 0,C 180,E1 -8928.966,E2 -8928.966} C_VEL
LIN {X 0,Y 438.651,Z 430.875,A -85,B 0,C 180,E1 -8930.639,E2 -8930.639} C_VEL
LIN {X 0,Y 438.904,Z 426.341,A -85,B 0,C 180,E1 -8932.116,E2 -8932.116} C_VEL
LIN {X 0,Y 439.326,Z 420.555,A -85,B 0,C 180,E1 -8933.573,E2 -8933.573} C_VEL
LIN {X 0,Y 439.816,Z 413.095,A -85,B 0,C 180,E1 -8935.052,E2 -8935.052} C_VEL
LIN {X 0,Y 440.358,Z 405.359,A -85,B 0,C 180,E1 -8936.287,E2 -8936.287} C_VEL
LIN {X 0,Y 441.02,Z 395.859,A -85,B 0,C 180,E1 -8937.524,E2 -8937.524} C_VEL
LIN {X 0,Y 441.621,Z 386.503,A -85,B 0,C 180,E1 -8938.516,E2 -8938.516} C_VEL
LIN {X 0,Y 442.309,Z 375.873,A -85,B 0,C 180,E1 -8939.426,E2 -8939.426} C_VEL
LIN {X 0,Y 442.873,Z 363.503,A -85,B 0,C 180,E1 -8940.253,E2 -8940.253} C_VEL
LIN {X 0,Y 443.347,Z 351.249,A -85,B 0,C 180,E1 -8940.867,E2 -8940.867} C_VEL
LIN {X 0,Y 443.708,Z 338.33,A -85,B 0,C 180,E1 -8941.311,E2 -8941.311} C_VEL
LIN {X 0,Y 443.896,Z 322.356,A -85,B 0,C 180,E1 -8941.63,E2 -8941.63} C_VEL
LIN {X 0,Y 444.775,Z 243.973,A -85,B 0,C 180,E1 -8942.92,E2 -8942.92} C_VEL
LIN {X 0,Y 441.099,Z 227.306,A -85,B 0,C 180,E1 -8943.404,E2 -8943.404} C_VEL
LIN {X 0,Y 440.972,Z 222.259,A -85,B 0,C 180,E1 -8944.481,E2 -8944.481} C_VEL
LIN {X 0,Y 439.379,Z 214.757,A -85,B 0,C 180,E1 -8946.229,E2 -8946.229} C_VEL
LIN {X 0,Y 439.416,Z 214.752,A -85,B 0,C 180,E1 -8949.852,E2 -8949.852} C_VEL
LIN {X 0,Y 439.391,Z 214.757,A -85,B 0,C 180,E1 -8952.629,E2 -8952.629} C_VEL
LIN {X 0,Y 439.389,Z 214.754,A -85,B 0,C 180,E1 -8956.032,E2 -8956.032} C_VEL
LIN {X 0,Y 439.383,Z 214.751,A -85,B 0,C 180,E1 -8959.02,E2 -8959.02} C_VEL
LIN {X 0,Y 439.372,Z 214.755,A -85,B 0,C 180,E1 -8961.604,E2 -8961.604} C_VEL
LIN {X 0,Y 439.381,Z 214.748,A -85,B 0,C 180,E1 -8964.843,E2 -8964.843} C_VEL
LIN {X 0,Y 439.353,Z 214.755,A -85,B 0,C 180,E1 -8968.138,E2 -8968.138} C_VEL
LIN {X 0,Y 439.403,Z 214.746,A -85,B 0,C 180,E1 -8971.326,E2 -8971.326} C_VEL
LIN {X 0,Y 439.382,Z 214.747,A -85,B 0,C 180,E1 -8974.414,E2 -8974.414} C_VEL
LIN {X 0,Y 439.357,Z 214.756,A -85,B 0,C 180,E1 -8977.424,E2 -8977.424} C_VEL
LIN {X 0,Y 439.416,Z 214.745,A -85,B 0,C 180,E1 -8980.662,E2 -8980.662} C_VEL
LIN {X 0,Y 439.449,Z 214.743,A -85,B 0,C 180,E1 -8984.224,E2 -8984.224} C_VEL
LIN {X 0,Y 439.456,Z 214.741,A -85,B 0,C 180,E1 -8988.001,E2 -8988.001} C_VEL
LIN {X 0,Y 439.52,Z 214.731,A -85,B 0,C 180,E1 -8991.726,E2 -8991.726} C_VEL
LIN {X 0,Y 439.597,Z 214.722,A -85,B 0,C 180,E1 -8994.496,E2 -8994.496} C_VEL
LIN {X 0,Y 439.602,Z 214.72,A -85,B 0,C 180,E1 -8998.168,E2 -8998.168} C_VEL
LIN {X 0,Y 439.73,Z 214.702,A -85,B 0,C 180,E1 -9000,E2 -9000} C_VEL
LIN {X 0,Y 439.609,Z 214.719,A -85,B 0,C 180,E1 -9002.749,E2 -9002.749} C_VEL
LIN {X 0,Y 439.568,Z 214.72,A -85,B 0,C 180,E1 -9006.426,E2 -9006.426} C_VEL
LIN {X 0,Y 439.47,Z 214.737,A -85,B 0,C 180,E1 -9009.203,E2 -9009.203} C_VEL
LIN {X 0,Y 439.479,Z 214.74,A -85,B 0,C 180,E1 -9012.727,E2 -9012.727} C_VEL
LIN {X 0,Y 439.42,Z 214.744,A -85,B 0,C 180,E1 -9016.349,E2 -9016.349} C_VEL
LIN {X 0,Y 439.377,Z 214.748,A -85,B 0,C 180,E1 -9019.628,E2 -9019.628} C_VEL
LIN {X 0,Y 439.337,Z 214.759,A -85,B 0,C 180,E1 -9022.577,E2 -9022.577} C_VEL
LIN {X 0,Y 439.353,Z 214.754,A -85,B 0,C 180,E1 -9025.588,E2 -9025.588} C_VEL
LIN {X 0,Y 439.376,Z 214.757,A -85,B 0,C 180,E1 -9028.677,E2 -9028.677} C_VEL
LIN {X 0,Y 439.343,Z 214.755,A -85,B 0,C 180,E1 -9032.03,E2 -9032.03} C_VEL
LIN {X 0,Y 439.372,Z 214.751,A -85,B 0,C 180,E1 -9035.341,E2 -9035.341} C_VEL
LIN {X 0,Y 439.346,Z 214.761,A -85,B 0,C 180,E1 -9038.599,E2 -9038.599} C_VEL
LIN {X 0,Y 439.368,Z 214.745,A -85,B 0,C 180,E1 -9041.257,E2 -9041.257} C_VEL
LIN {X 0,Y 439.365,Z 214.754,A -85,B 0,C 180,E1 -9044.734,E2 -9044.734} C_VEL
LIN {X 0,Y 439.373,Z 214.754,A -85,B 0,C 180,E1 -9047.796,E2 -9047.796} C_VEL
LIN {X 0,Y 439.355,Z 214.756,A -85,B 0,C 180,E1 -9051.404,E2 -9051.404} C_VEL
LIN {X 0,Y 439.394,Z 214.752,A -85,B 0,C 180,E1 -9054.845,E2 -9054.845} C_VEL
LIN {X 0,Y 439.369,Z 214.755,A -85,B 0,C 180,E1 -9058.141,E2 -9058.141} C_VEL
LIN {X 0,Y 439.407,Z 214.752,A -85,B 0,C 180,E1 -9061.605,E2 -9061.605} C_VEL
LIN {X 0,Y 439.477,Z 214.871,A -85,B 0,C 180,E1 -9062.312,E2 -9062.312} C_VEL
LIN {X 0,Y 442.164,Z 227.876,A -85,B 0,C 180,E1 -9064.958,E2 -9064.958} C_VEL
LIN {X 0,Y 442.383,Z 232.602,A -85,B 0,C 180,E1 -9065.853,E2 -9065.853} C_VEL
LIN {X 0,Y 441.289,Z 249.988,A -85,B 0,C 180,E1 -9069.002,E2 -9069.002} C_VEL
LIN {X 0,Y 440.568,Z 264.706,A -85,B 0,C 180,E1 -9071.635,E2 -9071.635} C_VEL
LIN {X 0,Y 444.321,Z 288.602,A -85,B 0,C 180,E1 -9072.223,E2 -9072.223} C_VEL
LIN {X 0,Y 443.548,Z 374.24,A -85,B 0,C 180,E1 -9073.665,E2 -9073.665} C_VEL
LIN {X 0,Y 443.017,Z 387.947,A -85,B 0,C 180,E1 -9074.089,E2 -9074.089} C_VEL
LIN {X 0,Y 442.359,Z 400.797,A -85,B 0,C 180,E1 -9074.685,E2 -9074.685} C_VEL
LIN {X 0,Y 441.725,Z 411.74,A -85,B 0,C 180,E1 -9075.37,E2 -9075.37} C_VEL
LIN {X 0,Y 441.027,Z 423.73,A -85,B 0,C 180,E1 -9076.333,E2 -9076.333} C_VEL
LIN {X 0,Y 440.398,Z 433.601,A -85,B 0,C 180,E1 -9077.324,E2 -9077.324} C_VEL
LIN {X 0,Y 439.82,Z 442.949,A -85,B 0,C 180,E1 -9078.478,E2 -9078.478} C_VEL
LIN {X 0,Y 439.175,Z 452.011,A -85,B 0,C 180,E1 -9079.861,E2 -9079.861} C_VEL
LIN {X 0,Y 438.821,Z 459.334,A -85,B 0,C 180,E1 -9081.248,E2 -9081.248} C_VEL
LIN {X 0,Y 438.526,Z 465.216,A -85,B 0,C 180,E1 -9082.633,E2 -9082.633} C_VEL
LIN {X 0,Y 438.347,Z 469.885,A -85,B 0,C 180,E1 -9084.025,E2 -9084.025} C_VEL
LIN {X 0,Y 438.341,Z 473.406,A -85,B 0,C 180,E1 -9085.401,E2 -9085.401} C_VEL
LIN {X 0,Y 438.286,Z 475.205,A -85,B 0,C 180,E1 -9086.321,E2 -9086.321} C_VEL
LIN {X 0,Y 438.371,Z 476.576,A -85,B 0,C 180,E1 -9087.242,E2 -9087.242} C_VEL
LIN {X 0,Y 438.309,Z 478.127,A -85,B 0,C 180,E1 -9089.08,E2 -9089.08} C_VEL
LIN {X 0,Y 438.315,Z 478.284,A -85,B 0,C 180,E1 -9089.998,E2 -9089.998} C_VEL
LIN {X 0,Y 438.318,Z 477.387,A -85,B 0,C 180,E1 -9091.836,E2 -9091.836} C_VEL
LIN {X 0,Y 438.371,Z 476.355,A -85,B 0,C 180,E1 -9092.755,E2 -9092.755} C_VEL
LIN {X 0,Y 438.292,Z 474.875,A -85,B 0,C 180,E1 -9093.676,E2 -9093.676} C_VEL
LIN {X 0,Y 438.406,Z 471.854,A -85,B 0,C 180,E1 -9095.056,E2 -9095.056} C_VEL
LIN {X 0,Y 438.447,Z 467.759,A -85,B 0,C 180,E1 -9096.44,E2 -9096.44} C_VEL
LIN {X 0,Y 438.653,Z 461.466,A -85,B 0,C 180,E1 -9098.057,E2 -9098.057} C_VEL
LIN {X 0,Y 438.911,Z 454.607,A -85,B 0,C 180,E1 -9099.444,E2 -9099.444} C_VEL
LIN {X 0,Y 439.355,Z 446.065,A -85,B 0,C 180,E1 -9100.831,E2 -9100.831} C_VEL
LIN {X 0,Y 439.876,Z 437.267,A -85,B 0,C 180,E1 -9101.985,E2 -9101.985} C_VEL
LIN {X 0,Y 440.505,Z 426.556,A -85,B 0,C 180,E1 -9103.126,E2 -9103.126} C_VEL
LIN {X 0,Y 441.092,Z 415.615,A -85,B 0,C 180,E1 -9104.06,E2 -9104.06} C_VEL
LIN {X 0,Y 441.705,Z 403.459,A -85,B 0,C 180,E1 -9104.863,E2 -9104.863} C_VEL
LIN {X 0,Y 442.295,Z 390.775,A -85,B 0,C 180,E1 -9105.492,E2 -9105.492} C_VEL
LIN {X 0,Y 442.71,Z 378.374,A -85,B 0,C 180,E1 -9105.919,E2 -9105.919} C_VEL
LIN {X 0,Y 443.008,Z 362.608,A -85,B 0,C 180,E1 -9106.234,E2 -9106.234} C_VEL
LIN {X 0,Y 443.591,Z 288.364,A -85,B 0,C 180,E1 -9107.443,E2 -9107.443} C_VEL
LIN {X 0,Y 440.253,Z 265.01,A -85,B 0,C 180,E1 -9107.977,E2 -9107.977} C_VEL
LIN {X 0,Y 440.992,Z 247.824,A -85,B 0,C 180,E1 -9111.009,E2 -9111.009} C_VEL
LIN {X 0,Y 441.875,Z 231.444,A -85,B 0,C 180,E1 -9113.923,E2 -9113.923} C_VEL
LIN {X 0,Y 441.794,Z 226.859,A -85,B 0,C 180,E1 -9114.76,E2 -9114.76} C_VEL
LIN {X 0,Y 439.51,Z 214.74,A -85,B 0,C 180,E1 -9117.107,E2 -9117.107} C_VEL
LIN {X 0,Y 439.346,Z 214.754,A -85,B 0,C 180,E1 -9120.785,E2 -9120.785} C_VEL
LIN {X 0,Y 439.37,Z 214.759,A -85,B 0,C 180,E1 -9124.04,E2 -9124.04} C_VEL
LIN {X 0,Y 439.329,Z 214.756,A -85,B 0,C 180,E1 -9126.883,E2 -9126.883} C_VEL
LIN {X 0,Y 439.379,Z 214.756,A -85,B 0,C 180,E1 -9129.845,E2 -9129.845} C_VEL
LIN {X 0,Y 439.356,Z 214.753,A -85,B 0,C 180,E1 -9132.623,E2 -9132.623} C_VEL
LIN {X 0,Y 439.374,Z 214.755,A -85,B 0,C 180,E1 -9136.03,E2 -9136.03} C_VEL
LIN {X 0,Y 439.37,Z 214.751,A -85,B 0,C 180,E1 -9139.018,E2 -9139.018} C_VEL
LIN {X 0,Y 439.36,Z 214.758,A -85,B 0,C 180,E1 -9141.601,E2 -9141.601} C_VEL
LIN {X 0,Y 439.364,Z 214.752,A -85,B 0,C 180,E1 -9144.84,E2 -9144.84} C_VEL
LIN {X 0,Y 439.334,Z 214.757,A -85,B 0,C 180,E1 -9148.136,E2 -9148.136} C_VEL
LIN {X 0,Y 439.385,Z 214.754,A -85,B 0,C 180,E1 -9151.324,E2 -9151.324} C_VEL
LIN {X 0,Y 439.371,Z 214.751,A -85,B 0,C 180,E1 -9154.413,E2 -9154.413} C_VEL
LIN {X 0,Y 439.34,Z 214.762,A -85,B 0,C 180,E1 -9157.423,E2 -9157.423} C_VEL
LIN {X 0,Y 439.395,Z 214.748,A -85,B 0,C 180,E1 -9160.661,E2 -9160.661} C_VEL
LIN {X 0,Y 439.427,Z 214.744,A -85,B 0,C 180,E1 -9164.223,E2 -9164.223} C_VEL
LIN {X 0,Y 439.463,Z 214.74,A -85,B 0,C 180,E1 -9168,E2 -9168} C_VEL
LIN {X 0,Y 439.503,Z 214.736,A -85,B 0,C 180,E1 -9171.725,E2 -9171.725} C_VEL
LIN {X 0,Y 439.578,Z 214.726,A -85,B 0,C 180,E1 -9174.495,E2 -9174.495} C_VEL
LIN {X 0,Y 439.582,Z 214.724,A -85,B 0,C 180,E1 -9178.167,E2 -9178.167} C_VEL
LIN {X 0,Y 439.709,Z 214.709,A -85,B 0,C 180,E1 -9180,E2 -9180} C_VEL
LIN {X 0,Y 439.588,Z 214.728,A -85,B 0,C 180,E1 -9182.749,E2 -9182.749} C_VEL
LIN {X 0,Y 439.56,Z 214.729,A -85,B 0,C 180,E1 -9186.426,E2 -9186.426} C_VEL
LIN {X 0,Y 439.45,Z 214.745,A -85,B 0,C 180,E1 -9189.202,E2 -9189.202} C_VEL
LIN {X 0,Y 439.454,Z 214.746,A -85,B 0,C 180,E1 -9192.727,E2 -9192.727} C_VEL
LIN {X 0,Y 439.411,Z 214.748,A -85,B 0,C 180,E1 -9196.356,E2 -9196.356} C_VEL
LIN {X 0,Y 439.354,Z 214.753,A -85,B 0,C 180,E1 -9199.628,E2 -9199.628} C_VEL
LIN {X 0,Y 439.319,Z 214.763,A -85,B 0,C 180,E1 -9202.578,E2 -9202.578} C_VEL
LIN {X 0,Y 439.359,Z 214.752,A -85,B 0,C 180,E1 -9205.587,E2 -9205.587} C_VEL
LIN {X 0,Y 439.374,Z 214.757,A -85,B 0,C 180,E1 -9208.676,E2 -9208.676} C_VEL
LIN {X 0,Y 439.327,Z 214.758,A -85,B 0,C 180,E1 -9212.033,E2 -9212.033} C_VEL
LIN {X 0,Y 439.356,Z 214.753,A -85,B 0,C 180,E1 -9215.343,E2 -9215.343} C_VEL
LIN {X 0,Y 439.334,Z 214.761,A -85,B 0,C 180,E1 -9218.6,E2 -9218.6} C_VEL
LIN {X 0,Y 439.354,Z 214.753,A -85,B 0,C 180,E1 -9221.26,E2 -9221.26} C_VEL
LIN {X 0,Y 439.367,Z 214.754,A -85,B 0,C 180,E1 -9224.733,E2 -9224.733} C_VEL
LIN {X 0,Y 439.367,Z 214.754,A -85,B 0,C 180,E1 -9227.799,E2 -9227.799} C_VEL
LIN {X 0,Y 439.41,Z 214.754,A -85,B 0,C 180,E1 -9230.232,E2 -9230.232} C_VEL
LIN {X 0,Y 439.351,Z 214.756,A -85,B 0,C 180,E1 -9233.716,E2 -9233.716} C_VEL
LIN {X 0,Y 439.352,Z 214.753,A -85,B 0,C 180,E1 -9237.058,E2 -9237.058} C_VEL
LIN {X 0,Y 439.364,Z 214.756,A -85,B 0,C 180,E1 -9240.278,E2 -9240.278} C_VEL
LIN {X 0,Y 439.413,Z 214.747,A -85,B 0,C 180,E1 -9243.4,E2 -9243.4} C_VEL
LIN {X 0,Y 439.371,Z 214.753,A -85,B 0,C 180,E1 -9246.433,E2 -9246.433} C_VEL
LIN {X 0,Y 439.376,Z 214.752,A -85,B 0,C 180,E1 -9249.4,E2 -9249.4} C_VEL
LIN {X 0,Y 439.394,Z 214.75,A -85,B 0,C 180,E1 -9252.311,E2 -9252.311} C_VEL
LIN {X 0,Y 439.438,Z 214.744,A -85,B 0,C 180,E1 -9255.177,E2 -9255.177} C_VEL
LIN {X 0,Y 439.477,Z 214.742,A -85,B 0,C 180,E1 -9258.004,E2 -9258.004} C_VEL
LIN {X 0,Y 439.5,Z 214.742,A -85,B 0,C 180,E1 -9261.728,E2 -9261.728} C_VEL
LIN {X 0,Y 439.59,Z 214.813,A -85,B 0,C 180,E1 -9264.469,E2 -9264.469} C_VEL
LIN {X 0,Y 440.644,Z 222.302,A -85,B 0,C 180,E1 -9266.115,E2 -9266.115} C_VEL
LIN {X 0,Y 440.617,Z 227.24,A -85,B 0,C 180,E1 -9267.145,E2 -9267.145} C_VEL
LIN {X 0,Y 442.015,Z 234.31,A -85,B 0,C 180,E1 -9267.315,E2 -9267.315} C_VEL
LIN {X 0,Y 442.339,Z 238.18,A -85,B 0,C 180,E1 -9267.391,E2 -9267.391} C_VEL
LIN {X 0,Y 442.018,Z 242.086,A -85,B 0,C 180,E1 -9267.445,E2 -9267.445} C_VEL
LIN {X 0,Y 440.214,Z 249.831,A -85,B 0,C 180,E1 -9267.509,E2 -9267.509} C_VEL
LIN {X 0,Y 438.017,Z 257.625,A -85,B 0,C 180,E1 -9267.56,E2 -9267.56} C_VEL
LIN {X 0,Y 437.005,Z 263.555,A -85,B 0,C 180,E1 -9267.624,E2 -9267.624} C_VEL
LIN {X 0,Y 436.916,Z 265.55,A -85,B 0,C 180,E1 -9267.654,E2 -9267.654} C_VEL
LIN {X 0,Y 436.178,Z 334.392,A -85,B 0,C 180,E1 -9268.807,E2 -9268.807} C_VEL
LIN {X 0,Y 435.818,Z 347.583,A -85,B 0,C 180,E1 -9269.207,E2 -9269.207} C_VEL
LIN {X 0,Y 435.44,Z 359.959,A -85,B 0,C 180,E1 -9269.77,E2 -9269.77} C_VEL
LIN {X 0,Y 434.996,Z 371.317,A -85,B 0,C 180,E1 -9270.464,E2 -9270.464} C_VEL
LIN {X 0,Y 434.305,Z 383.036,A -85,B 0,C 180,E1 -9271.392,E2 -9271.392} C_VEL
LIN {X 0,Y 433.686,Z 393.525,A -85,B 0,C 180,E1 -9272.439,E2 -9272.439} C_VEL
LIN {X 0,Y 433.183,Z 402.099,A -85,B 0,C 180,E1 -9273.489,E2 -9273.489} C_VEL
LIN {X 0,Y 432.666,Z 410.019,A -85,B 0,C 180,E1 -9274.66,E2 -9274.66} C_VEL
LIN {X 0,Y 432.195,Z 417.764,A -85,B 0,C 180,E1 -9276.068,E2 -9276.068} C_VEL
LIN {X 0,Y 431.922,Z 423.958,A -85,B 0,C 180,E1 -9277.48,E2 -9277.48} C_VEL
LIN {X 0,Y 431.618,Z 428.902,A -85,B 0,C 180,E1 -9278.899,E2 -9278.899} C_VEL
LIN {X 0,Y 431.431,Z 432.713,A -85,B 0,C 180,E1 -9280.323,E2 -9280.323} C_VEL
LIN {X 0,Y 431.298,Z 436.064,A -85,B 0,C 180,E1 -9282.124,E2 -9282.124} C_VEL
LIN {X 0,Y 431.193,Z 437.295,A -85,B 0,C 180,E1 -9283.191,E2 -9283.191} C_VEL
LIN {X 0,Y 431.15,Z 437.969,A -85,B 0,C 180,E1 -9284.153,E2 -9284.153} C_VEL
LIN {X 0,Y 431.158,Z 438.15,A -85,B 0,C 180,E1 -9285.906,E2 -9285.906} C_VEL
LIN {X 0,Y 431.162,Z 437.476,A -85,B 0,C 180,E1 -9287.062,E2 -9287.062} C_VEL
LIN {X 0,Y 431.253,Z 436.462,A -85,B 0,C 180,E1 -9288.037,E2 -9288.037} C_VEL
LIN {X 0,Y 431.408,Z 434.816,A -85,B 0,C 180,E1 -9289.115,E2 -9289.115} C_VEL
LIN {X 0,Y 431.571,Z 431.904,A -85,B 0,C 180,E1 -9290.494,E2 -9290.494} C_VEL
LIN {X 0,Y 431.817,Z 427.63,A -85,B 0,C 180,E1 -9291.983,E2 -9291.983} C_VEL
LIN {X 0,Y 432.242,Z 422.042,A -85,B 0,C 180,E1 -9293.475,E2 -9293.475} C_VEL
LIN {X 0,Y 432.762,Z 414.927,A -85,B 0,C 180,E1 -9294.975,E2 -9294.975} C_VEL
LIN {X 0,Y 433.326,Z 407.557,A -85,B 0,C 180,E1 -9296.228,E2 -9296.228} C_VEL
LIN {X 0,Y 433.979,Z 398.478,A -85,B 0,C 180,E1 -9297.485,E2 -9297.485} C_VEL
LIN {X 0,Y 434.677,Z 388.345,A -85,B 0,C 180,E1 -9298.618,E2 -9298.618} C_VEL
LIN {X 0,Y 435.477,Z 376.685,A -85,B 0,C 180,E1 -9299.657,E2 -9299.657} C_VEL
LIN {X 0,Y 436.086,Z 364.28,A -85,B 0,C 180,E1 -9300.507,E2 -9300.507} C_VEL
LIN {X 0,Y 436.605,Z 351.728,A -85,B 0,C 180,E1 -9301.149,E2 -9301.149} C_VEL
LIN {X 0,Y 436.993,Z 338.811,A -85,B 0,C 180,E1 -9301.602,E2 -9301.602} C_VEL
LIN {X 0,Y 437.217,Z 322.166,A -85,B 0,C 180,E1 -9301.938,E2 -9301.938} C_VEL
LIN {X 0,Y 438.226,Z 245.644,A -85,B 0,C 180,E1 -9303.212,E2 -9303.212} C_VEL
LIN {X 0,Y 434.229,Z 227.651,A -85,B 0,C 180,E1 -9303.746,E2 -9303.746} C_VEL
LIN {X 0,Y 433.865,Z 222.787,A -85,B 0,C 180,E1 -9304.818,E2 -9304.818} C_VEL
LIN {X 0,Y 432.334,Z 215.633,A -85,B 0,C 180,E1 -9306.501,E2 -9306.501} C_VEL
LIN {X 0,Y 432.355,Z 215.63,A -85,B 0,C 180,E1 -9309.34,E2 -9309.34} C_VEL
LIN {X 0,Y 432.363,Z 215.624,A -85,B 0,C 180,E1 -9311.791,E2 -9311.791} C_VEL
LIN {X 0,Y 432.366,Z 215.632,A -85,B 0,C 180,E1 -9314.34,E2 -9314.34} C_VEL
LIN {X 0,Y 432.351,Z 215.628,A -85,B 0,C 180,E1 -9317.008,E2 -9317.008} C_VEL
LIN {X 0,Y 432.34,Z 215.631,A -85,B 0,C 180,E1 -9319.816,E2 -9319.816} C_VEL
LIN {X 0,Y 432.298,Z 215.633,A -85,B 0,C 180,E1 -9323.021,E2 -9323.021} C_VEL
LIN {X 0,Y 432.34,Z 215.631,A -85,B 0,C 180,E1 -9325.995,E2 -9325.995} C_VEL
LIN {X 0,Y 432.373,Z 215.626,A -85,B 0,C 180,E1 -9329.743,E2 -9329.743} C_VEL
LIN {X 0,Y 432.377,Z 215.624,A -85,B 0,C 180,E1 -9333.372,E2 -9333.372} C_VEL
LIN {X 0,Y 432.351,Z 215.629,A -85,B 0,C 180,E1 -9336.023,E2 -9336.023} C_VEL
LIN {X 0,Y 432.349,Z 215.622,A -85,B 0,C 180,E1 -9339.046,E2 -9339.046} C_VEL
LIN {X 0,Y 432.353,Z 215.625,A -85,B 0,C 180,E1 -9342.01,E2 -9342.01} C_VEL
LIN {X 0,Y 432.375,Z 215.624,A -85,B 0,C 180,E1 -9344.926,E2 -9344.926} C_VEL
LIN {X 0,Y 432.432,Z 215.617,A -85,B 0,C 180,E1 -9347.803,E2 -9347.803} C_VEL
LIN {X 0,Y 432.465,Z 215.61,A -85,B 0,C 180,E1 -9351.59,E2 -9351.59} C_VEL
LIN {X 0,Y 432.574,Z 215.597,A -85,B 0,C 180,E1 -9354.406,E2 -9354.406} C_VEL
LIN {X 0,Y 432.573,Z 215.596,A -85,B 0,C 180,E1 -9358.138,E2 -9358.138} C_VEL
LIN {X 0,Y 432.701,Z 215.578,A -85,B 0,C 180,E1 -9360,E2 -9360} C_VEL
LIN {X 0,Y 432.561,Z 215.598,A -85,B 0,C 180,E1 -9362.794,E2 -9362.794} C_VEL
LIN {X 0,Y 432.557,Z 215.594,A -85,B 0,C 180,E1 -9365.595,E2 -9365.595} C_VEL
LIN {X 0,Y 432.437,Z 215.613,A -85,B 0,C 180,E1 -9368.411,E2 -9368.411} C_VEL
LIN {X 0,Y 432.455,Z 215.611,A -85,B 0,C 180,E1 -9372.197,E2 -9372.197} C_VEL
LIN {X 0,Y 432.404,Z 215.617,A -85,B 0,C 180,E1 -9376.04,E2 -9376.04} C_VEL
LIN {X 0,Y 432.362,Z 215.622,A -85,B 0,C 180,E1 -9379.486,E2 -9379.486} C_VEL
LIN {X 0,Y 432.291,Z 215.633,A -85,B 0,C 180,E1 -9382.966,E2 -9382.966} C_VEL
LIN {X 0,Y 432.311,Z 215.635,A -85,B 0,C 180,E1 -9385.004,E2 -9385.004} C_VEL
LIN {X 0,Y 432.322,Z 215.628,A -85,B 0,C 180,E1 -9388.128,E2 -9388.128} C_VEL
LIN {X 0,Y 432.295,Z 215.631,A -85,B 0,C 180,E1 -9391.348,E2 -9391.348} C_VEL
LIN {X 0,Y 432.309,Z 215.634,A -85,B 0,C 180,E1 -9394.68,E2 -9394.68} C_VEL
LIN {X 0,Y 432.313,Z 215.632,A -85,B 0,C 180,E1 -9398.153,E2 -9398.153} C_VEL
LIN {X 0,Y 432.311,Z 215.624,A -85,B 0,C 180,E1 -9401.602,E2 -9401.602} C_VEL
LIN {X 0,Y 432.321,Z 215.636,A -85,B 0,C 180,E1 -9404.349,E2 -9404.349} C_VEL
LIN {X 0,Y 432.307,Z 215.632,A -85,B 0,C 180,E1 -9407.018,E2 -9407.018} C_VEL
LIN {X 0,Y 432.282,Z 215.635,A -85,B 0,C 180,E1 -9409.829,E2 -9409.829} C_VEL
LIN {X 0,Y 432.299,Z 215.63,A -85,B 0,C 180,E1 -9413.023,E2 -9413.023} C_VEL
LIN {X 0,Y 432.355,Z 215.628,A -85,B 0,C 180,E1 -9415.998,E2 -9415.998} C_VEL
LIN {X 0,Y 432.344,Z 215.631,A -85,B 0,C 180,E1 -9419.491,E2 -9419.491} C_VEL
LIN {X 0,Y 432.412,Z 215.792,A -85,B 0,C 180,E1 -9422.012,E2 -9422.012} C_VEL
LIN {X 0,Y 435.169,Z 228.926,A -85,B 0,C 180,E1 -9424.744,E2 -9424.744} C_VEL
LIN {X 0,Y 435.551,Z 232.516,A -85,B 0,C 180,E1 -9425.45,E2 -9425.45} C_VEL
LIN {X 0,Y 434.356,Z 251.231,A -85,B 0,C 180,E1 -9428.899,E2 -9428.899} C_VEL
LIN {X 0,Y 433.676,Z 264.368,A -85,B 0,C 180,E1 -9431.291,E2 -9431.291} C_VEL
LIN {X 0,Y 437.503,Z 288.392,A -85,B 0,C 180,E1 -9431.899,E2 -9431.899} C_VEL
LIN {X 0,Y 437.688,Z 295.914,A -85,B 0,C 180,E1 -9432.037,E2 -9432.037} C_VEL
LIN {X 0,Y 436.835,Z 373.087,A -85,B 0,C 180,E1 -9433.347,E2 -9433.347} C_VEL
LIN {X 0,Y 436.377,Z 386.299,A -85,B 0,C 180,E1 -9433.75,E2 -9433.75} C_VEL
LIN {X 0,Y 435.67,Z 399.004,A -85,B 0,C 180,E1 -9434.324,E2 -9434.324} C_VEL
LIN {X 0,Y 434.943,Z 410.321,A -85,B 0,C 180,E1 -9435.017,E2 -9435.017} C_VEL
LIN {X 0,Y 434.242,Z 421.998,A -85,B 0,C 180,E1 -9435.95,E2 -9435.95} C_VEL
LIN {X 0,Y 433.497,Z 432.512,A -85,B 0,C 180,E1 -9437,E2 -9437} C_VEL
LIN {X 0,Y 432.948,Z 441.125,A -85,B 0,C 180,E1 -9438.055,E2 -9438.055} C_VEL
LIN {X 0,Y 432.329,Z 449.081,A -85,B 0,C 180,E1 -9439.225,E2 -9439.225} C_VEL
LIN {X 0,Y 431.875,Z 456.895,A -85,B 0,C 180,E1 -9440.634,E2 -9440.634} C_VEL
LIN {X 0,Y 431.534,Z 463.173,A -85,B 0,C 180,E1 -9442.042,E2 -9442.042} C_VEL
LIN {X 0,Y 431.318,Z 468.939,A -85,B 0,C 180,E1 -9443.697,E2 -9443.697} C_VEL
LIN {X 0,Y 431.269,Z 473.145,A -85,B 0,C 180,E1 -9445.325,E2 -9445.325} C_VEL
LIN {X 0,Y 431.192,Z 474.922,A -85,B 0,C 180,E1 -9446.261,E2 -9446.261} C_VEL
LIN {X 0,Y 431.279,Z 476.283,A -85,B 0,C 180,E1 -9447.196,E2 -9447.196} C_VEL
LIN {X 0,Y 431.222,Z 477.813,A -85,B 0,C 180,E1 -9449.065,E2 -9449.065} C_VEL
LIN {X 0,Y 431.226,Z 477.951,A -85,B 0,C 180,E1 -9449.998,E2 -9449.998} C_VEL
LIN {X 0,Y 431.241,Z 477.034,A -85,B 0,C 180,E1 -9451.866,E2 -9451.866} C_VEL
LIN {X 0,Y 431.279,Z 475.99,A -85,B 0,C 180,E1 -9452.8,E2 -9452.8} C_VEL
LIN {X 0,Y 431.198,Z 474.488,A -85,B 0,C 180,E1 -9453.736,E2 -9453.736} C_VEL
LIN {X 0,Y 431.312,Z 471.444,A -85,B 0,C 180,E1 -9455.14,E2 -9455.14} C_VEL
LIN {X 0,Y 431.374,Z 467.325,A -85,B 0,C 180,E1 -9456.546,E2 -9456.546} C_VEL
LIN {X 0,Y 431.584,Z 461.004,A -85,B 0,C 180,E1 -9458.189,E2 -9458.189} C_VEL
LIN {X 0,Y 431.871,Z 454.115,A -85,B 0,C 180,E1 -9459.599,E2 -9459.599} C_VEL
LIN {X 0,Y 432.343,Z 445.518,A -85,B 0,C 180,E1 -9461.009,E2 -9461.009} C_VEL
LIN {X 0,Y 432.846,Z 436.672,A -85,B 0,C 180,E1 -9462.183,E2 -9462.183} C_VEL
LIN {X 0,Y 433.521,Z 425.804,A -85,B 0,C 180,E1 -9463.352,E2 -9463.352} C_VEL
LIN {X 0,Y 434.134,Z 414.853,A -85,B 0,C 180,E1 -9464.29,E2 -9464.29} C_VEL
LIN {X 0,Y 434.792,Z 402.57,A -85,B 0,C 180,E1 -9465.105,E2 -9465.105} C_VEL
LIN {X 0,Y 435.359,Z 389.68,A -85,B 0,C 180,E1 -9465.745,E2 -9465.745} C_VEL
LIN {X 0,Y 435.859,Z 376.722,A -85,B 0,C 180,E1 -9466.177,E2 -9466.177} C_VEL
LIN {X 0,Y 436.117,Z 360.174,A -85,B 0,C 180,E1 -9466.497,E2 -9466.497} C_VEL
LIN {X 0,Y 436.725,Z 288.935,A -85,B 0,C 180,E1 -9467.673,E2 -9467.673} C_VEL
LIN {X 0,Y 433.287,Z 264.778,A -85,B 0,C 180,E1 -9468.221,E2 -9468.221} C_VEL
LIN {X 0,Y 434.191,Z 245.919,A -85,B 0,C 180,E1 -9471.603,E2 -9471.603} C_VEL
LIN {X 0,Y 434.992,Z 230.877,A -85,B 0,C 180,E1 -9474.326,E2 -9474.326} C_VEL
LIN {X 0,Y 434.271,Z 225.029,A -85,B 0,C 180,E1 -9475.442,E2 -9475.442} C_VEL
LIN {X 0,Y 432.455,Z 215.619,A -85,B 0,C 180,E1 -9477.325,E2 -9477.325} C_VEL
LIN {X 0,Y 432.333,Z 215.63,A -85,B 0,C 180,E1 -9480.506,E2 -9480.506} C_VEL
LIN {X 0,Y 432.342,Z 215.634,A -85,B 0,C 180,E1 -9484,E2 -9484} C_VEL
LIN {X 0,Y 432.302,Z 215.632,A -85,B 0,C 180,E1 -9487.193,E2 -9487.193} C_VEL
LIN {X 0,Y 432.31,Z 215.635,A -85,B 0,C 180,E1 -9490.175,E2 -9490.175} C_VEL
LIN {X 0,Y 432.292,Z 215.633,A -85,B 0,C 180,E1 -9493.057,E2 -9493.057} C_VEL
LIN {X 0,Y 432.334,Z 215.633,A -85,B 0,C 180,E1 -9495.657,E2 -9495.657} C_VEL
LIN {X 0,Y 432.343,Z 215.627,A -85,B 0,C 180,E1 -9498.388,E2 -9498.388} C_VEL
LIN {X 0,Y 432.32,Z 215.635,A -85,B 0,C 180,E1 -9501.848,E2 -9501.848} C_VEL
LIN {X 0,Y 432.304,Z 215.634,A -85,B 0,C 180,E1 -9505.319,E2 -9505.319} C_VEL
LIN {X 0,Y 432.284,Z 215.634,A -85,B 0,C 180,E1 -9508.651,E2 -9508.651} C_VEL
LIN {X 0,Y 432.341,Z 215.632,A -85,B 0,C 180,E1 -9511.366,E2 -9511.366} C_VEL
LIN {X 0,Y 432.326,Z 215.631,A -85,B 0,C 180,E1 -9513.965,E2 -9513.965} C_VEL
LIN {X 0,Y 432.289,Z 215.635,A -85,B 0,C 180,E1 -9517.034,E2 -9517.034} C_VEL
LIN {X 0,Y 432.336,Z 215.628,A -85,B 0,C 180,E1 -9520.039,E2 -9520.039} C_VEL
LIN {X 0,Y 432.375,Z 215.628,A -85,B 0,C 180,E1 -9523.515,E2 -9523.515} C_VEL
LIN {X 0,Y 432.397,Z 215.626,A -85,B 0,C 180,E1 -9527.187,E2 -9527.187} C_VEL
LIN {X 0,Y 432.406,Z 215.62,A -85,B 0,C 180,E1 -9530.646,E2 -9530.646} C_VEL
LIN {X 0,Y 432.554,Z 215.604,A -85,B 0,C 180,E1 -9533.469,E2 -9533.469} C_VEL
LIN {X 0,Y 432.553,Z 215.607,A -85,B 0,C 180,E1 -9537.206,E2 -9537.206} C_VEL
LIN {X 0,Y 432.679,Z 215.584,A -85,B 0,C 180,E1 -9540,E2 -9540} C_VEL
LIN {X 0,Y 432.54,Z 215.606,A -85,B 0,C 180,E1 -9542.794,E2 -9542.794} C_VEL
LIN {X 0,Y 432.516,Z 215.607,A -85,B 0,C 180,E1 -9546.531,E2 -9546.531} C_VEL
LIN {X 0,Y 432.394,Z 215.622,A -85,B 0,C 180,E1 -9549.354,E2 -9549.354} C_VEL
LIN {X 0,Y 432.395,Z 215.627,A -85,B 0,C 180,E1 -9552.812,E2 -9552.812} C_VEL
LIN {X 0,Y 432.374,Z 215.626,A -85,B 0,C 180,E1 -9556.485,E2 -9556.485} C_VEL
LIN {X 0,Y 432.29,Z 215.633,A -85,B 0,C 180,E1 -9559.962,E2 -9559.962} C_VEL
LIN {X 0,Y 432.273,Z 215.639,A -85,B 0,C 180,E1 -9562.966,E2 -9562.966} C_VEL
LIN {X 0,Y 432.319,Z 215.63,A -85,B 0,C 180,E1 -9566.035,E2 -9566.035} C_VEL
LIN {X 0,Y 432.299,Z 215.633,A -85,B 0,C 180,E1 -9569.19,E2 -9569.19} C_VEL
LIN {X 0,Y 432.282,Z 215.641,A -85,B 0,C 180,E1 -9572.446,E2 -9572.446} C_VEL
LIN {X 0,Y 432.307,Z 215.631,A -85,B 0,C 180,E1 -9575.635,E2 -9575.635} C_VEL
LIN {X 0,Y 432.297,Z 215.636,A -85,B 0,C 180,E1 -9578.716,E2 -9578.716} C_VEL
LIN {X 0,Y 432.299,Z 215.633,A -85,B 0,C 180,E1 -9581.801,E2 -9581.801} C_VEL
LIN {X 0,Y 432.303,Z 215.639,A -85,B 0,C 180,E1 -9584.351,E2 -9584.351} C_VEL
LIN {X 0,Y 432.291,Z 215.633,A -85,B 0,C 180,E1 -9587.02,E2 -9587.02} C_VEL
LIN {X 0,Y 432.314,Z 215.633,A -85,B 0,C 180,E1 -9589.823,E2 -9589.823} C_VEL
LIN {X 0,Y 432.283,Z 215.634,A -85,B 0,C 180,E1 -9593.026,E2 -9593.026} C_VEL
LIN {X 0,Y 432.338,Z 215.633,A -85,B 0,C 180,E1 -9596,E2 -9596} C_VEL
LIN {X 0,Y 432.329,Z 215.629,A -85,B 0,C 180,E1 -9599.493,E2 -9599.493} C_VEL
LIN {X 0,Y 432.375,Z 215.622,A -85,B 0,C 180,E1 -9602.932,E2 -9602.932} C_VEL
LIN {X 0,Y 432.354,Z 215.631,A -85,B 0,C 180,E1 -9606.027,E2 -9606.027} C_VEL
LIN {X 0,Y 432.338,Z 215.627,A -85,B 0,C 180,E1 -9609.049,E2 -9609.049} C_VEL
LIN {X 0,Y 432.35,Z 215.631,A -85,B 0,C 180,E1 -9612.013,E2 -9612.013} C_VEL
LIN {X 0,Y 432.385,Z 215.621,A -85,B 0,C 180,E1 -9614.929,E2 -9614.929} C_VEL
LIN {X 0,Y 432.453,Z 215.619,A -85,B 0,C 180,E1 -9617.806,E2 -9617.806} C_VEL
LIN {X 0,Y 432.46,Z 215.618,A -85,B 0,C 180,E1 -9621.592,E2 -9621.592} C_VEL
LIN {X 0,Y 432.584,Z 215.668,A -85,B 0,C 180,E1 -9624.291,E2 -9624.291} C_VEL
LIN {X 0,Y 433.69,Z 223.567,A -85,B 0,C 180,E1 -9626.053,E2 -9626.053} C_VEL
LIN {X 0,Y 433.644,Z 227.448,A -85,B 0,C 180,E1 -9626.878,E2 -9626.878} C_VEL
LIN {X 0,Y 437.139,Z 245.308,A -85,B 0,C 180,E1 -9627.32,E2 -9627.32} C_VEL
LIN {X 0,Y 436.916,Z 265.55,A -85,B 0,C 180,E1 -9627.654,E2 -9627.654} C_VEL
LIN {X 0,Y 436.223,Z 271.392,A -85,B 0,C 180,E1 -9627.728,E2 -9627.728} C_VEL
LIN {X 0,Y 430.413,Z 290.353,A -85,B 0,C 180,E1 -9627.84,E2 -9627.84} C_VEL
LIN {X 0,Y 429.734,Z 296.195,A -85,B 0,C 180,E1 -9627.915,E2 -9627.915} C_VEL
LIN {X 0,Y 429.235,Z 335.816,A -85,B 0,C 180,E1 -9628.606,E2 -9628.606} C_VEL
LIN {X 0,Y 428.906,Z 349.054,A -85,B 0,C 180,E1 -9629.031,E2 -9629.031} C_VEL
LIN {X 0,Y 428.523,Z 361.327,A -85,B 0,C 180,E1 -9629.614,E2 -9629.614} C_VEL
LIN {X 0,Y 427.994,Z 372.888,A -85,B 0,C 180,E1 -9630.354,E2 -9630.354} C_VEL
LIN {X 0,Y 427.295,Z 384.356,A -85,B 0,C 180,E1 -9631.297,E2 -9631.297} C_VEL
LIN {X 0,Y 426.659,Z 394.675,A -85,B 0,C 180,E1 -9632.362,E2 -9632.362} C_VEL
LIN {X 0,Y 426.085,Z 403.949,A -85,B 0,C 180,E1 -9633.548,E2 -9633.548} C_VEL
LIN {X 0,Y 425.544,Z 412.932,A -85,B 0,C 180,E1 -9634.975,E2 -9634.975} C_VEL
LIN {X 0,Y 425.092,Z 420.189,A -85,B 0,C 180,E1 -9636.408,E2 -9636.408} C_VEL
LIN {X 0,Y 424.82,Z 425.092,A -85,B 0,C 180,E1 -9637.606,E2 -9637.606} C_VEL
LIN {X 0,Y 424.506,Z 429.871,A -85,B 0,C 180,E1 -9639.05,E2 -9639.05} C_VEL
LIN {X 0,Y 424.336,Z 433.522,A -85,B 0,C 180,E1 -9640.498,E2 -9640.498} C_VEL
LIN {X 0,Y 424.219,Z 436.508,A -85,B 0,C 180,E1 -9642.193,E2 -9642.193} C_VEL
LIN {X 0,Y 424.099,Z 437.808,A -85,B 0,C 180,E1 -9643.415,E2 -9643.415} C_VEL
LIN {X 0,Y 424.053,Z 438.41,A -85,B 0,C 180,E1 -9644.395,E2 -9644.395} C_VEL
LIN {X 0,Y 424.089,Z 438.461,A -85,B 0,C 180,E1 -9646.019,E2 -9646.019} C_VEL
LIN {X 0,Y 424.091,Z 437.623,A -85,B 0,C 180,E1 -9647.355,E2 -9647.355} C_VEL
LIN {X 0,Y 424.201,Z 436.517,A -85,B 0,C 180,E1 -9648.348,E2 -9648.348} C_VEL
LIN {X 0,Y 424.404,Z 433.98,A -85,B 0,C 180,E1 -9649.845,E2 -9649.845} C_VEL
LIN {X 0,Y 424.653,Z 430.332,A -85,B 0,C 180,E1 -9651.352,E2 -9651.352} C_VEL
LIN {X 0,Y 424.978,Z 425.44,A -85,B 0,C 180,E1 -9652.869,E2 -9652.869} C_VEL
LIN {X 0,Y 425.493,Z 419.144,A -85,B 0,C 180,E1 -9654.389,E2 -9654.389} C_VEL
LIN {X 0,Y 426.121,Z 411.18,A -85,B 0,C 180,E1 -9655.916,E2 -9655.916} C_VEL
LIN {X 0,Y 426.813,Z 402.562,A -85,B 0,C 180,E1 -9657.231,E2 -9657.231} C_VEL
LIN {X 0,Y 427.547,Z 392.54,A -85,B 0,C 180,E1 -9658.469,E2 -9658.469} C_VEL
LIN {X 0,Y 428.311,Z 382.297,A -85,B 0,C 180,E1 -9659.488,E2 -9659.488} C_VEL
LIN {X 0,Y 429.057,Z 371.19,A -85,B 0,C 180,E1 -9660.365,E2 -9660.365} C_VEL
LIN {X 0,Y 429.596,Z 359.488,A -85,B 0,C 180,E1 -9661.086,E2 -9661.086} C_VEL
LIN {X 0,Y 430.095,Z 346.44,A -85,B 0,C 180,E1 -9661.674,E2 -9661.674} C_VEL
LIN {X 0,Y 430.399,Z 333.6,A -85,B 0,C 180,E1 -9662.048,E2 -9662.048} C_VEL
LIN {X 0,Y 431.554,Z 246.276,A -85,B 0,C 180,E1 -9663.542,E2 -9663.542} C_VEL
LIN {X 0,Y 427.563,Z 228.994,A -85,B 0,C 180,E1 -9664.063,E2 -9664.063} C_VEL
LIN {X 0,Y 427.363,Z 227.871,A -85,B 0,C 180,E1 -9664.128,E2 -9664.128} C_VEL
LIN {X 0,Y 426.694,Z 223.157,A -85,B 0,C 180,E1 -9665.202,E2 -9665.202} C_VEL
LIN {X 0,Y 425.297,Z 216.511,A -85,B 0,C 180,E1 -9666.798,E2 -9666.798} C_VEL
LIN {X 0,Y 425.299,Z 216.513,A -85,B 0,C 180,E1 -9670.124,E2 -9670.124} C_VEL
LIN {X 0,Y 425.305,Z 216.509,A -85,B 0,C 180,E1 -9673.358,E2 -9673.358} C_VEL
LIN {X 0,Y 425.318,Z 216.506,A -85,B 0,C 180,E1 -9676.637,E2 -9676.637} C_VEL
LIN {X 0,Y 425.293,Z 216.508,A -85,B 0,C 180,E1 -9679.874,E2 -9679.874} C_VEL
LIN {X 0,Y 425.269,Z 216.51,A -85,B 0,C 180,E1 -9682.486,E2 -9682.486} C_VEL
LIN {X 0,Y 425.289,Z 216.507,A -85,B 0,C 180,E1 -9685.816,E2 -9685.816} C_VEL
LIN {X 0,Y 425.279,Z 216.506,A -85,B 0,C 180,E1 -9689.236,E2 -9689.236} C_VEL
LIN {X 0,Y 425.328,Z 216.501,A -85,B 0,C 180,E1 -9692.441,E2 -9692.441} C_VEL
LIN {X 0,Y 425.33,Z 216.499,A -85,B 0,C 180,E1 -9695.601,E2 -9695.601} C_VEL
LIN {X 0,Y 425.294,Z 216.5,A -85,B 0,C 180,E1 -9698.682,E2 -9698.682} C_VEL
LIN {X 0,Y 425.308,Z 216.506,A -85,B 0,C 180,E1 -9701.702,E2 -9701.702} C_VEL
LIN {X 0,Y 425.329,Z 216.501,A -85,B 0,C 180,E1 -9704.67,E2 -9704.67} C_VEL
LIN {X 0,Y 425.385,Z 216.494,A -85,B 0,C 180,E1 -9707.598,E2 -9707.598} C_VEL
LIN {X 0,Y 425.416,Z 216.489,A -85,B 0,C 180,E1 -9711.45,E2 -9711.45} C_VEL
LIN {X 0,Y 425.531,Z 216.474,A -85,B 0,C 180,E1 -9714.313,E2 -9714.313} C_VEL
LIN {X 0,Y 425.542,Z 216.472,A -85,B 0,C 180,E1 -9718.107,E2 -9718.107} C_VEL
LIN {X 0,Y 425.671,Z 216.453,A -85,B 0,C 180,E1 -9720,E2 -9720} C_VEL
LIN {X 0,Y 425.515,Z 216.476,A -85,B 0,C 180,E1 -9722.84,E2 -9722.84} C_VEL
LIN {X 0,Y 425.513,Z 216.471,A -85,B 0,C 180,E1 -9725.688,E2 -9725.688} C_VEL
LIN {X 0,Y 425.382,Z 216.493,A -85,B 0,C 180,E1 -9728.552,E2 -9728.552} C_VEL
LIN {X 0,Y 425.404,Z 216.49,A -85,B 0,C 180,E1 -9732.402,E2 -9732.402} C_VEL
LIN {X 0,Y 425.362,Z 216.495,A -85,B 0,C 180,E1 -9736.313,E2 -9736.313} C_VEL
LIN {X 0,Y 425.304,Z 216.501,A -85,B 0,C 180,E1 -9739.636,E2 -9739.636} C_VEL
LIN {X 0,Y 425.265,Z 216.511,A -85,B 0,C 180,E1 -9742.34,E2 -9742.34} C_VEL
LIN {X 0,Y 425.288,Z 216.509,A -85,B 0,C 180,E1 -9744.655,E2 -9744.655} C_VEL
LIN {X 0,Y 425.248,Z 216.508,A -85,B 0,C 180,E1 -9747.565,E2 -9747.565} C_VEL
LIN {X 0,Y 425.27,Z 216.509,A -85,B 0,C 180,E1 -9750.762,E2 -9750.762} C_VEL
LIN {X 0,Y 425.274,Z 216.51,A -85,B 0,C 180,E1 -9754.285,E2 -9754.285} C_VEL
LIN {X 0,Y 425.26,Z 216.508,A -85,B 0,C 180,E1 -9757.697,E2 -9757.697} C_VEL
LIN {X 0,Y 425.252,Z 216.508,A -85,B 0,C 180,E1 -9760.519,E2 -9760.519} C_VEL
LIN {X 0,Y 425.243,Z 216.511,A -85,B 0,C 180,E1 -9763.352,E2 -9763.352} C_VEL
LIN {X 0,Y 425.246,Z 216.514,A -85,B 0,C 180,E1 -9766.651,E2 -9766.651} C_VEL
LIN {X 0,Y 425.236,Z 216.512,A -85,B 0,C 180,E1 -9769.869,E2 -9769.869} C_VEL
LIN {X 0,Y 425.27,Z 216.508,A -85,B 0,C 180,E1 -9772.49,E2 -9772.49} C_VEL
LIN {X 0,Y 425.303,Z 216.506,A -85,B 0,C 180,E1 -9775.819,E2 -9775.819} C_VEL
LIN {X 0,Y 425.288,Z 216.51,A -85,B 0,C 180,E1 -9779.24,E2 -9779.24} C_VEL
LIN {X 0,Y 425.358,Z 216.605,A -85,B 0,C 180,E1 -9781.674,E2 -9781.674} C_VEL
LIN {X 0,Y 428.189,Z 229.991,A -85,B 0,C 180,E1 -9784.52,E2 -9784.52} C_VEL
LIN {X 0,Y 428.679,Z 233.788,A -85,B 0,C 180,E1 -9785.288,E2 -9785.288} C_VEL
LIN {X 0,Y 427.501,Z 251.146,A -85,B 0,C 180,E1 -9788.544,E2 -9788.544} C_VEL
LIN {X 0,Y 426.777,Z 263.899,A -85,B 0,C 180,E1 -9790.908,E2 -9790.908} C_VEL
LIN {X 0,Y 430.479,Z 286.578,A -85,B 0,C 180,E1 -9791.521,E2 -9791.521} C_VEL
LIN {X 0,Y 431.079,Z 292.007,A -85,B 0,C 180,E1 -9791.647,E2 -9791.647} C_VEL
LIN {X 0,Y 430.124,Z 373.062,A -85,B 0,C 180,E1 -9793.049,E2 -9793.049} C_VEL
LIN {X 0,Y 429.643,Z 386.17,A -85,B 0,C 180,E1 -9793.457,E2 -9793.457} C_VEL
LIN {X 0,Y 428.91,Z 398.261,A -85,B 0,C 180,E1 -9794.009,E2 -9794.009} C_VEL
LIN {X 0,Y 428.109,Z 410.496,A -85,B 0,C 180,E1 -9794.772,E2 -9794.772} C_VEL
LIN {X 0,Y 427.336,Z 422.074,A -85,B 0,C 180,E1 -9795.718,E2 -9795.718} C_VEL
LIN {X 0,Y 426.556,Z 432.518,A -85,B 0,C 180,E1 -9796.785,E2 -9796.785} C_VEL
LIN {X 0,Y 425.975,Z 441.075,A -85,B 0,C 180,E1 -9797.856,E2 -9797.856} C_VEL
LIN {X 0,Y 425.331,Z 448.985,A -85,B 0,C 180,E1 -9799.045,E2 -9799.045} C_VEL
LIN {X 0,Y 424.819,Z 456.739,A -85,B 0,C 180,E1 -9800.477,E2 -9800.477} C_VEL
LIN {X 0,Y 424.489,Z 462.979,A -85,B 0,C 180,E1 -9801.909,E2 -9801.909} C_VEL
LIN {X 0,Y 424.257,Z 467.954,A -85,B 0,C 180,E1 -9803.34,E2 -9803.34} C_VEL
LIN {X 0,Y 424.197,Z 471.809,A -85,B 0,C 180,E1 -9804.771,E2 -9804.771} C_VEL
LIN {X 0,Y 424.103,Z 474.642,A -85,B 0,C 180,E1 -9806.198,E2 -9806.198} C_VEL
LIN {X 0,Y 424.174,Z 475.991,A -85,B 0,C 180,E1 -9807.149,E2 -9807.149} C_VEL
LIN {X 0,Y 424.166,Z 476.942,A -85,B 0,C 180,E1 -9808.1,E2 -9808.1} C_VEL
LIN {X 0,Y 424.139,Z 477.497,A -85,B 0,C 180,E1 -9809.049,E2 -9809.049} C_VEL
LIN {X 0,Y 424.14,Z 477.618,A -85,B 0,C 180,E1 -9809.998,E2 -9809.998} C_VEL
LIN {X 0,Y 424.165,Z 476.682,A -85,B 0,C 180,E1 -9811.897,E2 -9811.897} C_VEL
LIN {X 0,Y 424.19,Z 475.624,A -85,B 0,C 180,E1 -9812.847,E2 -9812.847} C_VEL
LIN {X 0,Y 424.108,Z 474.102,A -85,B 0,C 180,E1 -9813.799,E2 -9813.799} C_VEL
LIN {X 0,Y 424.22,Z 471.034,A -85,B 0,C 180,E1 -9815.226,E2 -9815.226} C_VEL
LIN {X 0,Y 424.297,Z 466.887,A -85,B 0,C 180,E1 -9816.656,E2 -9816.656} C_VEL
LIN {X 0,Y 424.509,Z 460.532,A -85,B 0,C 180,E1 -9818.327,E2 -9818.327} C_VEL
LIN {X 0,Y 424.839,Z 453.606,A -85,B 0,C 180,E1 -9819.76,E2 -9819.76} C_VEL
LIN {X 0,Y 425.22,Z 446.528,A -85,B 0,C 180,E1 -9820.954,E2 -9820.954} C_VEL
LIN {X 0,Y 425.779,Z 438.001,A -85,B 0,C 180,E1 -9822.146,E2 -9822.146} C_VEL
LIN {X 0,Y 426.443,Z 427.448,A -85,B 0,C 180,E1 -9823.337,E2 -9823.337} C_VEL
LIN {X 0,Y 427.118,Z 415.555,A -85,B 0,C 180,E1 -9824.408,E2 -9824.408} C_VEL
LIN {X 0,Y 427.814,Z 403.586,A -85,B 0,C 180,E1 -9825.236,E2 -9825.236} C_VEL
LIN {X 0,Y 428.43,Z 391.123,A -85,B 0,C 180,E1 -9825.884,E2 -9825.884} C_VEL
LIN {X 0,Y 428.918,Z 378.271,A -85,B 0,C 180,E1 -9826.354,E2 -9826.354} C_VEL
LIN {X 0,Y 429.221,Z 364.644,A -85,B 0,C 180,E1 -9826.648,E2 -9826.648} C_VEL
LIN {X 0,Y 429.849,Z 289.47,A -85,B 0,C 180,E1 -9827.911,E2 -9827.911} C_VEL
LIN {X 0,Y 426.306,Z 264.393,A -85,B 0,C 180,E1 -9828.499,E2 -9828.499} C_VEL
LIN {X 0,Y 427.355,Z 243.972,A -85,B 0,C 180,E1 -9832.221,E2 -9832.221} C_VEL
LIN {X 0,Y 428.03,Z 231.658,A -85,B 0,C 180,E1 -9834.489,E2 -9834.489} C_VEL
LIN {X 0,Y 426.991,Z 224.673,A -85,B 0,C 180,E1 -9835.856,E2 -9835.856} C_VEL
LIN {X 0,Y 425.404,Z 216.497,A -85,B 0,C 180,E1 -9837.507,E2 -9837.507} C_VEL
LIN {X 0,Y 425.273,Z 216.507,A -85,B 0,C 180,E1 -9840.812,E2 -9840.812} C_VEL
LIN {X 0,Y 425.294,Z 216.509,A -85,B 0,C 180,E1 -9844.284,E2 -9844.284} C_VEL
LIN {X 0,Y 425.259,Z 216.513,A -85,B 0,C 180,E1 -9847.69,E2 -9847.69} C_VEL
LIN {X 0,Y 425.256,Z 216.51,A -85,B 0,C 180,E1 -9850.516,E2 -9850.516} C_VEL
LIN {X 0,Y 425.232,Z 216.514,A -85,B 0,C 180,E1 -9853.347,E2 -9853.347} C_VEL
LIN {X 0,Y 425.285,Z 216.506,A -85,B 0,C 180,E1 -9856.637,E2 -9856.637} C_VEL
LIN {X 0,Y 425.282,Z 216.512,A -85,B 0,C 180,E1 -9859.872,E2 -9859.872} C_VEL
LIN {X 0,Y 425.253,Z 216.51,A -85,B 0,C 180,E1 -9862.483,E2 -9862.483} C_VEL
LIN {X 0,Y 425.271,Z 216.513,A -85,B 0,C 180,E1 -9865.814,E2 -9865.814} C_VEL
LIN {X 0,Y 425.26,Z 216.512,A -85,B 0,C 180,E1 -9869.234,E2 -9869.234} C_VEL
LIN {X 0,Y 425.309,Z 216.502,A -85,B 0,C 180,E1 -9872.439,E2 -9872.439} C_VEL
LIN {X 0,Y 425.314,Z 216.508,A -85,B 0,C 180,E1 -9875.6,E2 -9875.6} C_VEL
LIN {X 0,Y 425.276,Z 216.507,A -85,B 0,C 180,E1 -9878.68,E2 -9878.68} C_VEL
LIN {X 0,Y 425.286,Z 216.509,A -85,B 0,C 180,E1 -9881.7,E2 -9881.7} C_VEL
LIN {X 0,Y 425.309,Z 216.503,A -85,B 0,C 180,E1 -9884.669,E2 -9884.669} C_VEL
LIN {X 0,Y 425.383,Z 216.497,A -85,B 0,C 180,E1 -9887.597,E2 -9887.597} C_VEL
LIN {X 0,Y 425.417,Z 216.494,A -85,B 0,C 180,E1 -9891.449,E2 -9891.449} C_VEL
LIN {X 0,Y 425.532,Z 216.475,A -85,B 0,C 180,E1 -9894.313,E2 -9894.313} C_VEL
LIN {X 0,Y 425.522,Z 216.476,A -85,B 0,C 180,E1 -9898.107,E2 -9898.107} C_VEL
LIN {X 0,Y 425.65,Z 216.46,A -85,B 0,C 180,E1 -9900,E2 -9900} C_VEL
LIN {X 0,Y 425.494,Z 216.485,A -85,B 0,C 180,E1 -9902.84,E2 -9902.84} C_VEL
LIN {X 0,Y 425.474,Z 216.485,A -85,B 0,C 180,E1 -9906.639,E2 -9906.639} C_VEL
LIN {X 0,Y 425.353,Z 216.498,A -85,B 0,C 180,E1 -9909.51,E2 -9909.51} C_VEL
LIN {X 0,Y 425.354,Z 216.504,A -85,B 0,C 180,E1 -9912.911,E2 -9912.911} C_VEL
LIN {X 0,Y 425.321,Z 216.506,A -85,B 0,C 180,E1 -9916.61,E2 -9916.61} C_VEL
LIN {X 0,Y 425.281,Z 216.506,A -85,B 0,C 180,E1 -9919.637,E2 -9919.637} C_VEL
LIN {X 0,Y 425.242,Z 216.514,A -85,B 0,C 180,E1 -9922.341,E2 -9922.341} C_VEL
LIN {X 0,Y 425.25,Z 216.51,A -85,B 0,C 180,E1 -9925.448,E2 -9925.448} C_VEL
LIN {X 0,Y 425.288,Z 216.512,A -85,B 0,C 180,E1 -9928.635,E2 -9928.635} C_VEL
LIN {X 0,Y 425.223,Z 216.514,A -85,B 0,C 180,E1 -9931.93,E2 -9931.93} C_VEL
LIN {X 0,Y 425.262,Z 216.508,A -85,B 0,C 180,E1 -9935.339,E2 -9935.339} C_VEL
LIN {X 0,Y 425.257,Z 216.511,A -85,B 0,C 180,E1 -9938.903,E2 -9938.903} C_VEL
LIN {X 0,Y 425.256,Z 216.512,A -85,B 0,C 180,E1 -9941.961,E2 -9941.961} C_VEL
LIN {X 0,Y 425.255,Z 216.509,A -85,B 0,C 180,E1 -9945.287,E2 -9945.287} C_VEL
LIN {X 0,Y 425.247,Z 216.513,A -85,B 0,C 180,E1 -9948.625,E2 -9948.625} C_VEL
LIN {X 0,Y 425.287,Z 216.505,A -85,B 0,C 180,E1 -9951.106,E2 -9951.106} C_VEL
LIN {X 0,Y 425.278,Z 216.508,A -85,B 0,C 180,E1 -9954.668,E2 -9954.668} C_VEL
LIN {X 0,Y 425.246,Z 216.518,A -85,B 0,C 180,E1 -9958.077,E2 -9958.077} C_VEL
LIN {X 0,Y 425.314,Z 216.503,A -85,B 0,C 180,E1 -9961.371,E2 -9961.371} C_VEL
LIN {X 0,Y 425.339,Z 216.501,A -85,B 0,C 180,E1 -9963.509,E2 -9963.509} C_VEL
LIN {X 0,Y 425.272,Z 216.508,A -85,B 0,C 180,E1 -9966.637,E2 -9966.637} C_VEL
LIN {X 0,Y 425.284,Z 216.511,A -85,B 0,C 180,E1 -9969.698,E2 -9969.698} C_VEL
LIN {X 0,Y 425.324,Z 216.501,A -85,B 0,C 180,E1 -9972.7,E2 -9972.7} C_VEL
LIN {X 0,Y 425.339,Z 216.505,A -85,B 0,C 180,E1 -9975.653,E2 -9975.653} C_VEL
LIN {X 0,Y 425.344,Z 216.498,A -85,B 0,C 180,E1 -9978.567,E2 -9978.567} C_VEL
LIN {X 0,Y 425.404,Z 216.495,A -85,B 0,C 180,E1 -9981.452,E2 -9981.452} C_VEL
LIN {X 0,Y 425.537,Z 216.615,A -85,B 0,C 180,E1 -9984.137,E2 -9984.137} C_VEL
LIN {X 0,Y 426.723,Z 224.823,A -85,B 0,C 180,E1 -9985.988,E2 -9985.988} C_VEL
LIN {X 0,Y 426.693,Z 227.764,A -85,B 0,C 180,E1 -9986.623,E2 -9986.623} C_VEL
LIN {X 0,Y 430.316,Z 245.982,A -85,B 0,C 180,E1 -9987.076,E2 -9987.076} C_VEL
LIN {X 0,Y 429.734,Z 296.195,A -85,B 0,C 180,E1 -9987.915,E2 -9987.915} C_VEL
LIN {X 0,Y 429.061,Z 302.034,A -85,B 0,C 180,E1 -9987.991,E2 -9987.991} C_VEL
LIN {X 0,Y 423.241,Z 320.987,A -85,B 0,C 180,E1 -9988.11,E2 -9988.11} C_VEL
LIN {X 0,Y 422.508,Z 326.828,A -85,B 0,C 180,E1 -9988.186,E2 -9988.186} C_VEL
LIN {X 0,Y 422.288,Z 340.704,A -85,B 0,C 180,E1 -9988.498,E2 -9988.498} C_VEL
LIN {X 0,Y 421.944,Z 353.02,A -85,B 0,C 180,E1 -9988.963,E2 -9988.963} C_VEL
LIN {X 0,Y 421.501,Z 365.153,A -85,B 0,C 180,E1 -9989.608,E2 -9989.608} C_VEL
LIN {X 0,Y 420.84,Z 377.526,A -85,B 0,C 180,E1 -9990.48,E2 -9990.48} C_VEL
LIN {X 0,Y 420.069,Z 389.262,A -85,B 0,C 180,E1 -9991.559,E2 -9991.559} C_VEL
LIN {X 0,Y 419.469,Z 398.705,A -85,B 0,C 180,E1 -9992.642,E2 -9992.642} C_VEL
LIN {X 0,Y 418.829,Z 407.351,A -85,B 0,C 180,E1 -9993.85,E2 -9993.85} C_VEL
LIN {X 0,Y 418.327,Z 415.716,A -85,B 0,C 180,E1 -9995.303,E2 -9995.303} C_VEL
LIN {X 0,Y 417.945,Z 422.458,A -85,B 0,C 180,E1 -9996.761,E2 -9996.761} C_VEL
LIN {X 0,Y 417.602,Z 427.861,A -85,B 0,C 180,E1 -9998.225,E2 -9998.225} C_VEL
LIN {X 0,Y 417.332,Z 432.086,A -85,B 0,C 180,E1 -9999.696,E2 -9999.696} C_VEL
LIN {X 0,Y 417.22,Z 434.322,A -85,B 0,C 180,E1 -10000.679,E2 -10000.679} C_VEL
LIN {X 0,Y 417.122,Z 436.921,A -85,B 0,C 180,E1 -10002.252,E2 -10002.252} C_VEL
LIN {X 0,Y 417,Z 438.32,A -85,B 0,C 180,E1 -10003.648,E2 -10003.648} C_VEL
LIN {X 0,Y 416.96,Z 438.805,A -85,B 0,C 180,E1 -10004.645,E2 -10004.645} C_VEL
LIN {X 0,Y 417.012,Z 438.767,A -85,B 0,C 180,E1 -10006.131,E2 -10006.131} C_VEL
LIN {X 0,Y 417.034,Z 437.757,A -85,B 0,C 180,E1 -10007.659,E2 -10007.659} C_VEL
LIN {X 0,Y 417.3,Z 435.32,A -85,B 0,C 180,E1 -10009.417,E2 -10009.417} C_VEL
LIN {X 0,Y 417.564,Z 431.411,A -85,B 0,C 180,E1 -10011.215,E2 -10011.215} C_VEL
LIN {X 0,Y 417.881,Z 426.782,A -85,B 0,C 180,E1 -10012.756,E2 -10012.756} C_VEL
LIN {X 0,Y 418.407,Z 420.775,A -85,B 0,C 180,E1 -10014.3,E2 -10014.3} C_VEL
LIN {X 0,Y 419.062,Z 413.111,A -85,B 0,C 180,E1 -10015.851,E2 -10015.851} C_VEL
LIN {X 0,Y 419.803,Z 404.609,A -85,B 0,C 180,E1 -10017.233,E2 -10017.233} C_VEL
LIN {X 0,Y 420.515,Z 395.432,A -85,B 0,C 180,E1 -10018.444,E2 -10018.444} C_VEL
LIN {X 0,Y 421.376,Z 384.409,A -85,B 0,C 180,E1 -10019.605,E2 -10019.605} C_VEL
LIN {X 0,Y 422.162,Z 373.582,A -85,B 0,C 180,E1 -10020.513,E2 -10020.513} C_VEL
LIN {X 0,Y 422.807,Z 361.677,A -85,B 0,C 180,E1 -10021.294,E2 -10021.294} C_VEL
LIN {X 0,Y 423.355,Z 348.737,A -85,B 0,C 180,E1 -10021.912,E2 -10021.912} C_VEL
LIN {X 0,Y 423.672,Z 336.058,A -85,B 0,C 180,E1 -10022.322,E2 -10022.322} C_VEL
LIN {X 0,Y 424.875,Z 247.01,A -85,B 0,C 180,E1 -10023.885,E2 -10023.885} C_VEL
LIN {X 0,Y 421.104,Z 230.652,A -85,B 0,C 180,E1 -10024.39,E2 -10024.39} C_VEL
LIN {X 0,Y 420.437,Z 228.335,A -85,B 0,C 180,E1 -10024.48,E2 -10024.48} C_VEL
LIN {X 0,Y 418.568,Z 218.915,A -85,B 0,C 180,E1 -10026.712,E2 -10026.712} C_VEL
LIN {X 0,Y 418.263,Z 217.386,A -85,B 0,C 180,E1 -10027.1,E2 -10027.1} C_VEL
LIN {X 0,Y 418.255,Z 217.387,A -85,B 0,C 180,E1 -10029.679,E2 -10029.679} C_VEL
LIN {X 0,Y 418.274,Z 217.384,A -85,B 0,C 180,E1 -10032.328,E2 -10032.328} C_VEL
LIN {X 0,Y 418.262,Z 217.384,A -85,B 0,C 180,E1 -10035.113,E2 -10035.113} C_VEL
LIN {X 0,Y 418.277,Z 217.382,A -85,B 0,C 180,E1 -10037.772,E2 -10037.772} C_VEL
LIN {X 0,Y 418.248,Z 217.386,A -85,B 0,C 180,E1 -10041.558,E2 -10041.558} C_VEL
LIN {X 0,Y 418.241,Z 217.381,A -85,B 0,C 180,E1 -10045.158,E2 -10045.158} C_VEL
LIN {X 0,Y 418.226,Z 217.388,A -85,B 0,C 180,E1 -10047.471,E2 -10047.471} C_VEL
LIN {X 0,Y 418.255,Z 217.379,A -85,B 0,C 180,E1 -10050.893,E2 -10050.893} C_VEL
LIN {X 0,Y 418.248,Z 217.382,A -85,B 0,C 180,E1 -10054.095,E2 -10054.095} C_VEL
LIN {X 0,Y 418.253,Z 217.386,A -85,B 0,C 180,E1 -10057.536,E2 -10057.536} C_VEL
LIN {X 0,Y 418.293,Z 217.378,A -85,B 0,C 180,E1 -10060.365,E2 -10060.365} C_VEL
LIN {X 0,Y 418.301,Z 217.375,A -85,B 0,C 180,E1 -10063.404,E2 -10063.404} C_VEL
LIN {X 0,Y 418.32,Z 217.374,A -85,B 0,C 180,E1 -10067,E2 -10067} C_VEL
LIN {X 0,Y 418.314,Z 217.374,A -85,B 0,C 180,E1 -10070.328,E2 -10070.328} C_VEL
LIN {X 0,Y 418.472,Z 217.355,A -85,B 0,C 180,E1 -10073.249,E2 -10073.249} C_VEL
LIN {X 0,Y 418.313,Z 217.378,A -85,B 0,C 180,E1 -10075.182,E2 -10075.182} C_VEL
LIN {X 0,Y 418.512,Z 217.347,A -85,B 0,C 180,E1 -10078.076,E2 -10078.076} C_VEL
LIN {X 0,Y 418.641,Z 217.329,A -85,B 0,C 180,E1 -10080,E2 -10080} C_VEL
LIN {X 0,Y 418.47,Z 217.353,A -85,B 0,C 180,E1 -10082.888,E2 -10082.888} C_VEL
LIN {X 0,Y 418.472,Z 217.347,A -85,B 0,C 180,E1 -10085.784,E2 -10085.784} C_VEL
LIN {X 0,Y 418.352,Z 217.37,A -85,B 0,C 180,E1 -10088.696,E2 -10088.696} C_VEL
LIN {X 0,Y 418.306,Z 217.374,A -85,B 0,C 180,E1 -10091.632,E2 -10091.632} C_VEL
